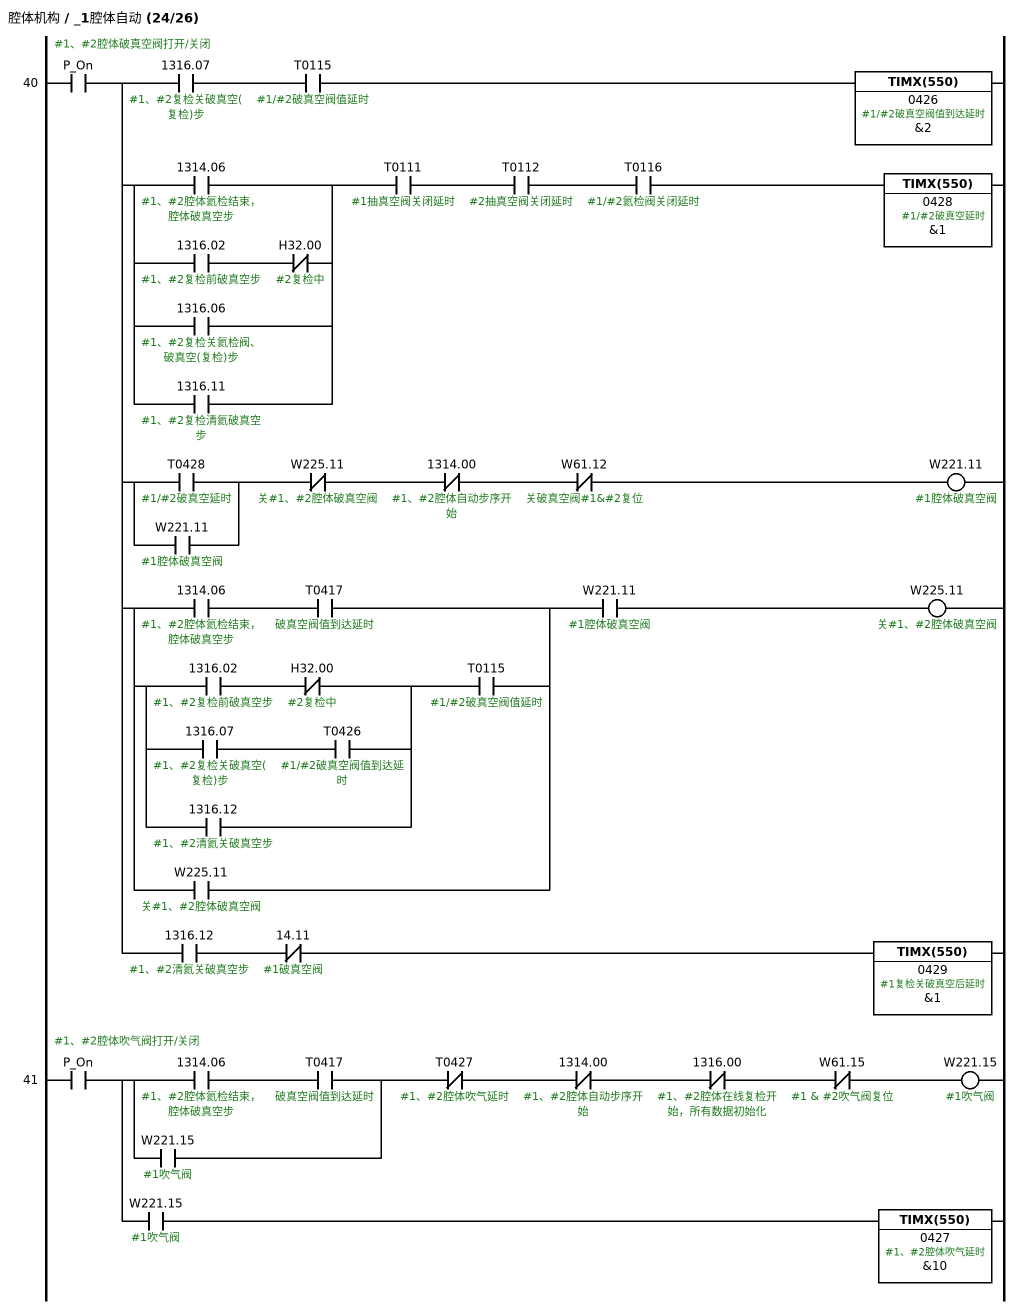
; [picture p264: 腔体机构 / _1腔体自动, rungs 40-41]
; rung 40: #1、#2腔体破真空阀打开/关闭
LD P_On
OUT TR0
AND 1316.07  ; #1、#2复检关破真空(复检)步
AND T0115  ; #1/#2破真空阀值延时
TIMX(550) 0426 &2  ; #1/#2破真空阀值到达延时
LD TR0
LD 1314.06  ; #1、#2腔体氦检结束，腔体破真空步
LD 1316.02  ; #1、#2复检前破真空步
ANDNOT H32.00  ; #2复检中
ORLD
OR 1316.06  ; #1、#2复检关氦检阀、破真空(复检)步
OR 1316.11  ; #1、#2复检清氦破真空步
ANDLD
AND T0111  ; #1抽真空阀关闭延时
AND T0112  ; #2抽真空阀关闭延时
AND T0116  ; #1/#2氦检阀关闭延时
TIMX(550) 0428 &1  ; #1/#2破真空延时
LD TR0
LD T0428  ; #1/#2破真空延时
OR W221.11  ; #1腔体破真空阀
ANDLD
ANDNOT W225.11  ; 关#1、#2腔体破真空阀
ANDNOT 1314.00  ; #1、#2腔体自动步序开始
ANDNOT W61.12  ; 关破真空阀#1&#2复位
OUT W221.11  ; #1腔体破真空阀
LD TR0
LD 1314.06  ; #1、#2腔体氦检结束，腔体破真空步
AND T0417  ; 破真空阀值到达延时
LD 1316.02  ; #1、#2复检前破真空步
ANDNOT H32.00  ; #2复检中
LD 1316.07  ; #1、#2复检关破真空(复检)步
AND T0426  ; #1/#2破真空阀值到达延时
ORLD
OR 1316.12  ; #1、#2清氦关破真空步
AND T0115  ; #1/#2破真空阀值延时
ORLD
OR W225.11  ; 关#1、#2腔体破真空阀
ANDLD
AND W221.11  ; #1腔体破真空阀
OUT W225.11  ; 关#1、#2腔体破真空阀
LD TR0
AND 1316.12  ; #1、#2清氦关破真空步
ANDNOT 14.11  ; #1破真空阀
TIMX(550) 0429 &1  ; #1复检关破真空后延时
; rung 41: #1、#2腔体吹气阀打开/关闭
LD P_On
OUT TR0
LD 1314.06  ; #1、#2腔体氦检结束，腔体破真空步
AND T0417  ; 破真空阀值到达延时
OR W221.15  ; #1吹气阀
ANDLD
ANDNOT T0427  ; #1、#2腔体吹气延时
ANDNOT 1314.00  ; #1、#2腔体自动步序开始
ANDNOT 1316.00  ; #1、#2腔体在线复检开始，所有数据初始化
ANDNOT W61.15  ; #1 & #2吹气阀复位
OUT W221.15  ; #1吹气阀
LD TR0
AND W221.15  ; #1吹气阀
TIMX(550) 0427 &10  ; #1、#2腔体吹气延时

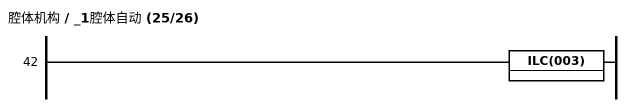
; rung 42
ILC(003)

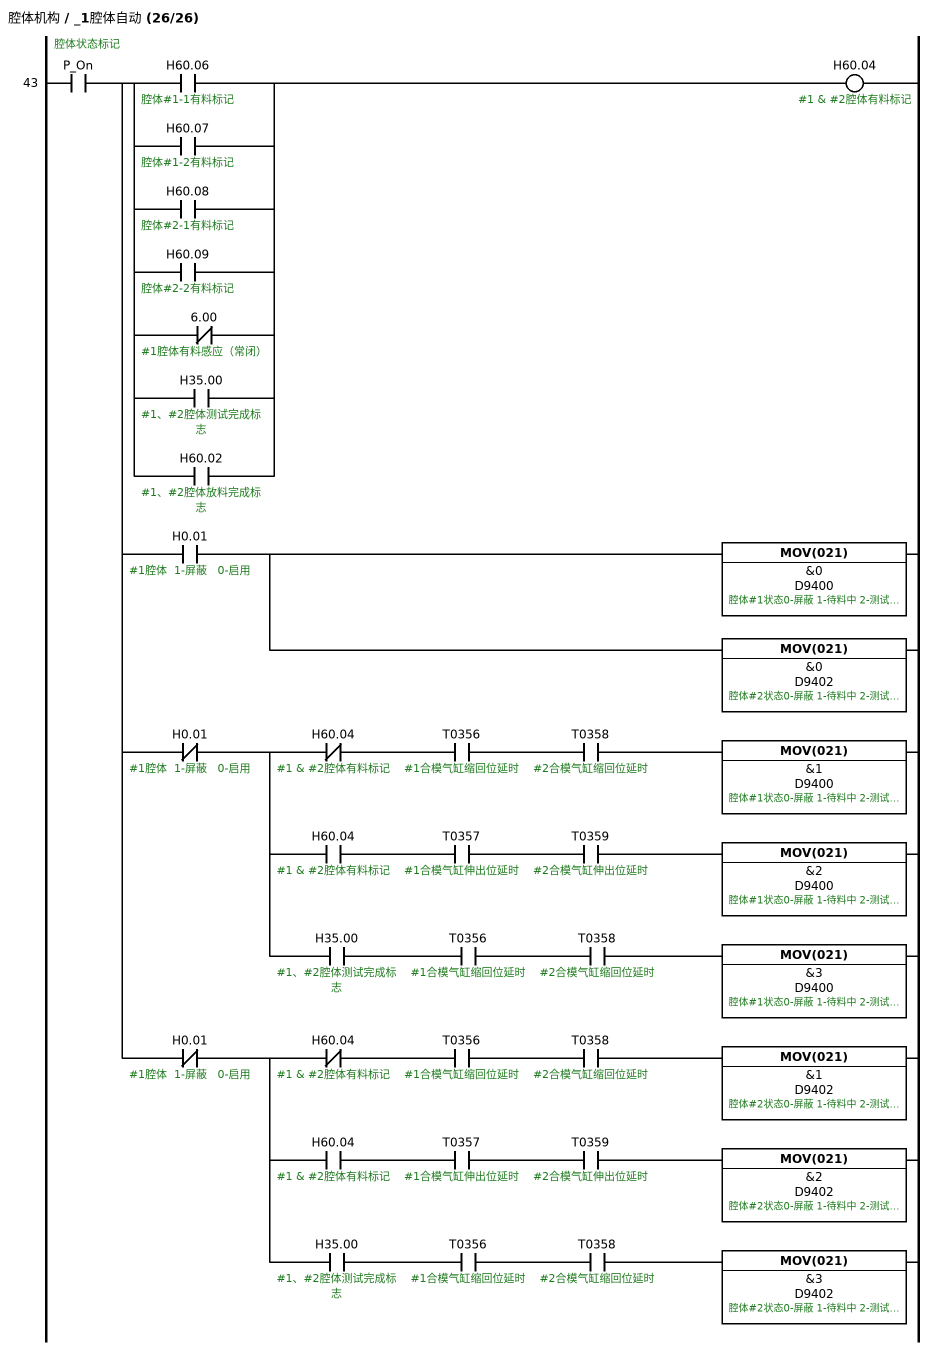
; rung 43: 腔体状态标记
LD P_On
OUT TR0
LD H60.06  ; 腔体#1-1有料标记
OR H60.07  ; 腔体#1-2有料标记
OR H60.08  ; 腔体#2-1有料标记
OR H60.09  ; 腔体#2-2有料标记
ORNOT 6.00  ; #1腔体有料感应（常闭）
OR H35.00  ; #1、#2腔体测试完成标志
OR H60.02  ; #1、#2腔体放料完成标志
ANDLD
OUT H60.04  ; #1 & #2腔体有料标记
LD TR0
AND H0.01  ; #1腔体  1-屏蔽   0-启用
MOV(021) &0 D9400  ; 腔体#1状态0-屏蔽 1-待料中 2-测试中 3-测试完成 4-在线复检
MOV(021) &0 D9402  ; 腔体#2状态0-屏蔽 1-待料中 2-测试中 3-测试完成 4-在线复检
LD TR0
ANDNOT H0.01  ; #1腔体  1-屏蔽   0-启用
OUT TR1
ANDNOT H60.04  ; #1 & #2腔体有料标记
AND T0356  ; #1合模气缸缩回位延时
AND T0358  ; #2合模气缸缩回位延时
MOV(021) &1 D9400  ; 腔体#1状态0-屏蔽 1-待料中 2-测试中 3-测试完成 4-在线复检
LD TR1
AND H60.04  ; #1 & #2腔体有料标记
AND T0357  ; #1合模气缸伸出位延时
AND T0359  ; #2合模气缸伸出位延时
MOV(021) &2 D9400  ; 腔体#1状态0-屏蔽 1-待料中 2-测试中 3-测试完成 4-在线复检
LD TR1
AND H35.00  ; #1、#2腔体测试完成标志
AND T0356  ; #1合模气缸缩回位延时
AND T0358  ; #2合模气缸缩回位延时
MOV(021) &3 D9400  ; 腔体#1状态0-屏蔽 1-待料中 2-测试中 3-测试完成 4-在线复检
LD TR0
ANDNOT H0.01  ; #1腔体  1-屏蔽   0-启用
OUT TR0
ANDNOT H60.04  ; #1 & #2腔体有料标记
AND T0356  ; #1合模气缸缩回位延时
AND T0358  ; #2合模气缸缩回位延时
MOV(021) &1 D9402  ; 腔体#2状态0-屏蔽 1-待料中 2-测试中 3-测试完成 4-在线复检
LD TR0
AND H60.04  ; #1 & #2腔体有料标记
AND T0357  ; #1合模气缸伸出位延时
AND T0359  ; #2合模气缸伸出位延时
MOV(021) &2 D9402  ; 腔体#2状态0-屏蔽 1-待料中 2-测试中 3-测试完成 4-在线复检
LD TR0
AND H35.00  ; #1、#2腔体测试完成标志
AND T0356  ; #1合模气缸缩回位延时
AND T0358  ; #2合模气缸缩回位延时
MOV(021) &3 D9402  ; 腔体#2状态0-屏蔽 1-待料中 2-测试中 3-测试完成 4-在线复检

### Section _2腔体自动

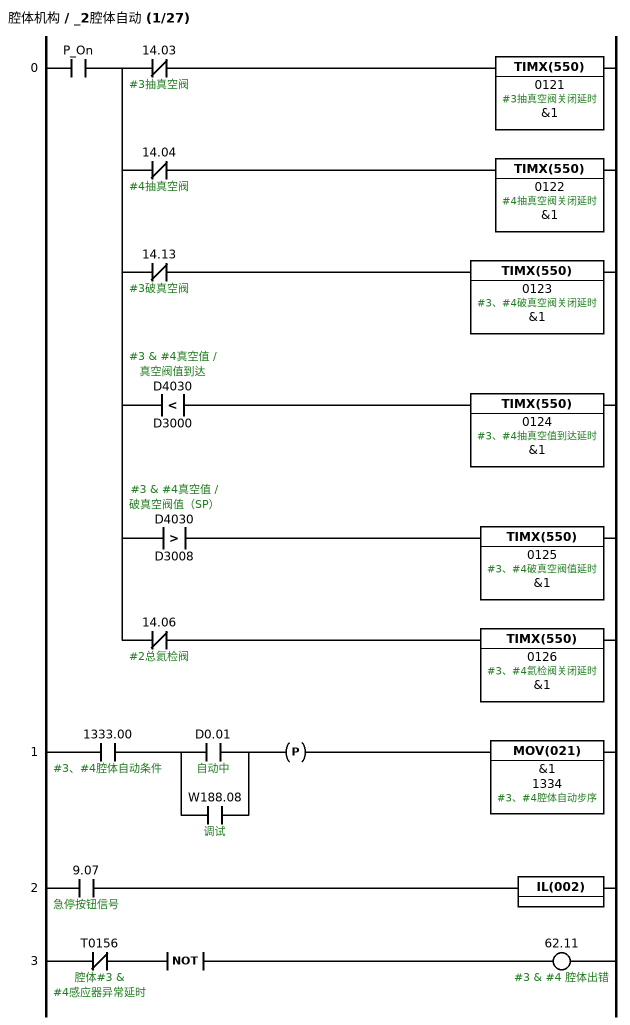
; rung 0
LD P_On
OUT TR0
ANDNOT 14.03  ; #3抽真空阀
TIMX(550) 0121 &1  ; #3抽真空阀关闭延时
LD TR0
ANDNOT 14.04  ; #4抽真空阀
TIMX(550) 0122 &1  ; #4抽真空阀关闭延时
LD TR0
ANDNOT 14.13  ; #3破真空阀
TIMX(550) 0123 &1  ; #3、#4破真空阀关闭延时
LD TR0
AND<F(331) D4030 D3000  ; #3 & #4真空值, 真空阀值到达
TIMX(550) 0124 &1  ; #3、#4抽真空值到达延时
LD TR0
AND>F(333) D4030 D3008  ; #3 & #4真空值, 破真空阀值（SP）
TIMX(550) 0125 &1  ; #3、#4破真空阀值延时
LD TR0
ANDNOT 14.06  ; #2总氦检阀
TIMX(550) 0126 &1  ; #3、#4氦检阀关闭延时
; rung 1
LD 1333.00  ; #3、#4腔体自动条件
LD D0.01  ; 自动中
OR W188.08  ; 调试
ANDLD
UP(521)
MOV(021) &1 1334  ; #3、#4腔体自动步序
; rung 2
LD 9.07  ; 急停按钮信号
IL(002)
; rung 3
LDNOT T0156  ; 腔体#3 & #4感应器异常延时
NOT(520)
OUT 62.11  ; #3 & #4 腔体出错

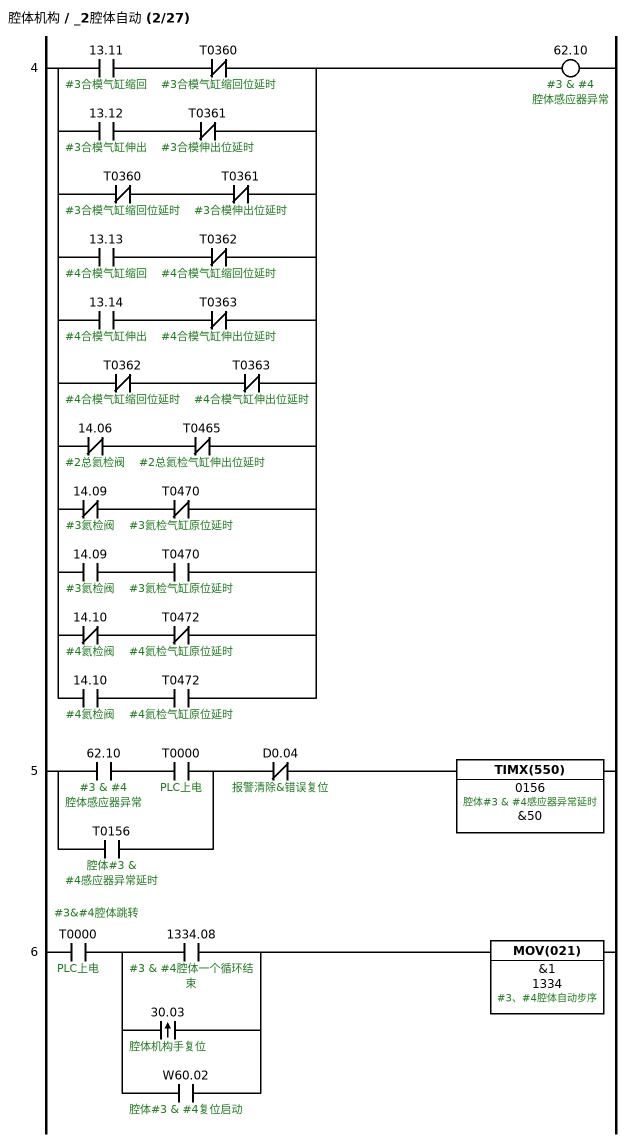
; rung 4
LD 13.11  ; #3合模气缸缩回
ANDNOT T0360  ; #3合模气缸缩回位延时
LD 13.12  ; #3合模气缸伸出
ANDNOT T0361  ; #3合模伸出位延时
ORLD
LDNOT T0360  ; #3合模气缸缩回位延时
ANDNOT T0361  ; #3合模伸出位延时
ORLD
LD 13.13  ; #4合模气缸缩回
ANDNOT T0362  ; #4合模气缸缩回位延时
ORLD
LD 13.14  ; #4合模气缸伸出
ANDNOT T0363  ; #4合模气缸伸出位延时
ORLD
LDNOT T0362  ; #4合模气缸缩回位延时
ANDNOT T0363  ; #4合模气缸伸出位延时
ORLD
LDNOT 14.06  ; #2总氦检阀
ANDNOT T0465  ; #2总氦检气缸伸出位延时
ORLD
LDNOT 14.09  ; #3氦检阀
ANDNOT T0470  ; #3氦检气缸原位延时
ORLD
LD 14.09  ; #3氦检阀
AND T0470  ; #3氦检气缸原位延时
ORLD
LDNOT 14.10  ; #4氦检阀
ANDNOT T0472  ; #4氦检气缸原位延时
ORLD
LD 14.10  ; #4氦检阀
AND T0472  ; #4氦检气缸原位延时
ORLD
OUT 62.10  ; #3 & #4 腔体感应器异常
; rung 5
LD 62.10  ; #3 & #4 腔体感应器异常
AND T0000  ; PLC上电
OR T0156  ; 腔体#3 & #4感应器异常延时
ANDNOT D0.04  ; 报警清除&错误复位
TIMX(550) 0156 &50  ; 腔体#3 & #4感应器异常延时
; rung 6: #3&#4腔体跳转
LD T0000  ; PLC上电
LD 1334.08  ; #3 & #4腔体一个循环结束
@OR 30.03  ; 腔体机构手复位
OR W60.02  ; 腔体#3 & #4复位启动
ANDLD
MOV(021) &1 1334  ; #3、#4腔体自动步序

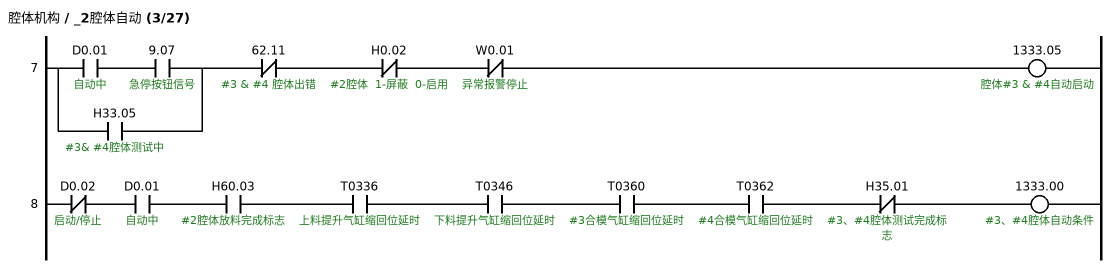
; rung 7
LD D0.01  ; 自动中
AND 9.07  ; 急停按钮信号
OR H33.05  ; #3& #4腔体测试中
ANDNOT 62.11  ; #3 & #4 腔体出错
ANDNOT H0.02  ; #2腔体  1-屏蔽  0-启用
ANDNOT W0.01  ; 异常报警停止
OUT 1333.05  ; 腔体#3 & #4自动启动
; rung 8
LDNOT D0.02  ; 启动/停止
AND D0.01  ; 自动中
AND H60.03  ; #2腔体放料完成标志
AND T0336  ; 上料提升气缸缩回位延时
AND T0346  ; 下料提升气缸缩回位延时
AND T0360  ; #3合模气缸缩回位延时
AND T0362  ; #4合模气缸缩回位延时
ANDNOT H35.01  ; #3、#4腔体测试完成标志
OUT 1333.00  ; #3、#4腔体自动条件

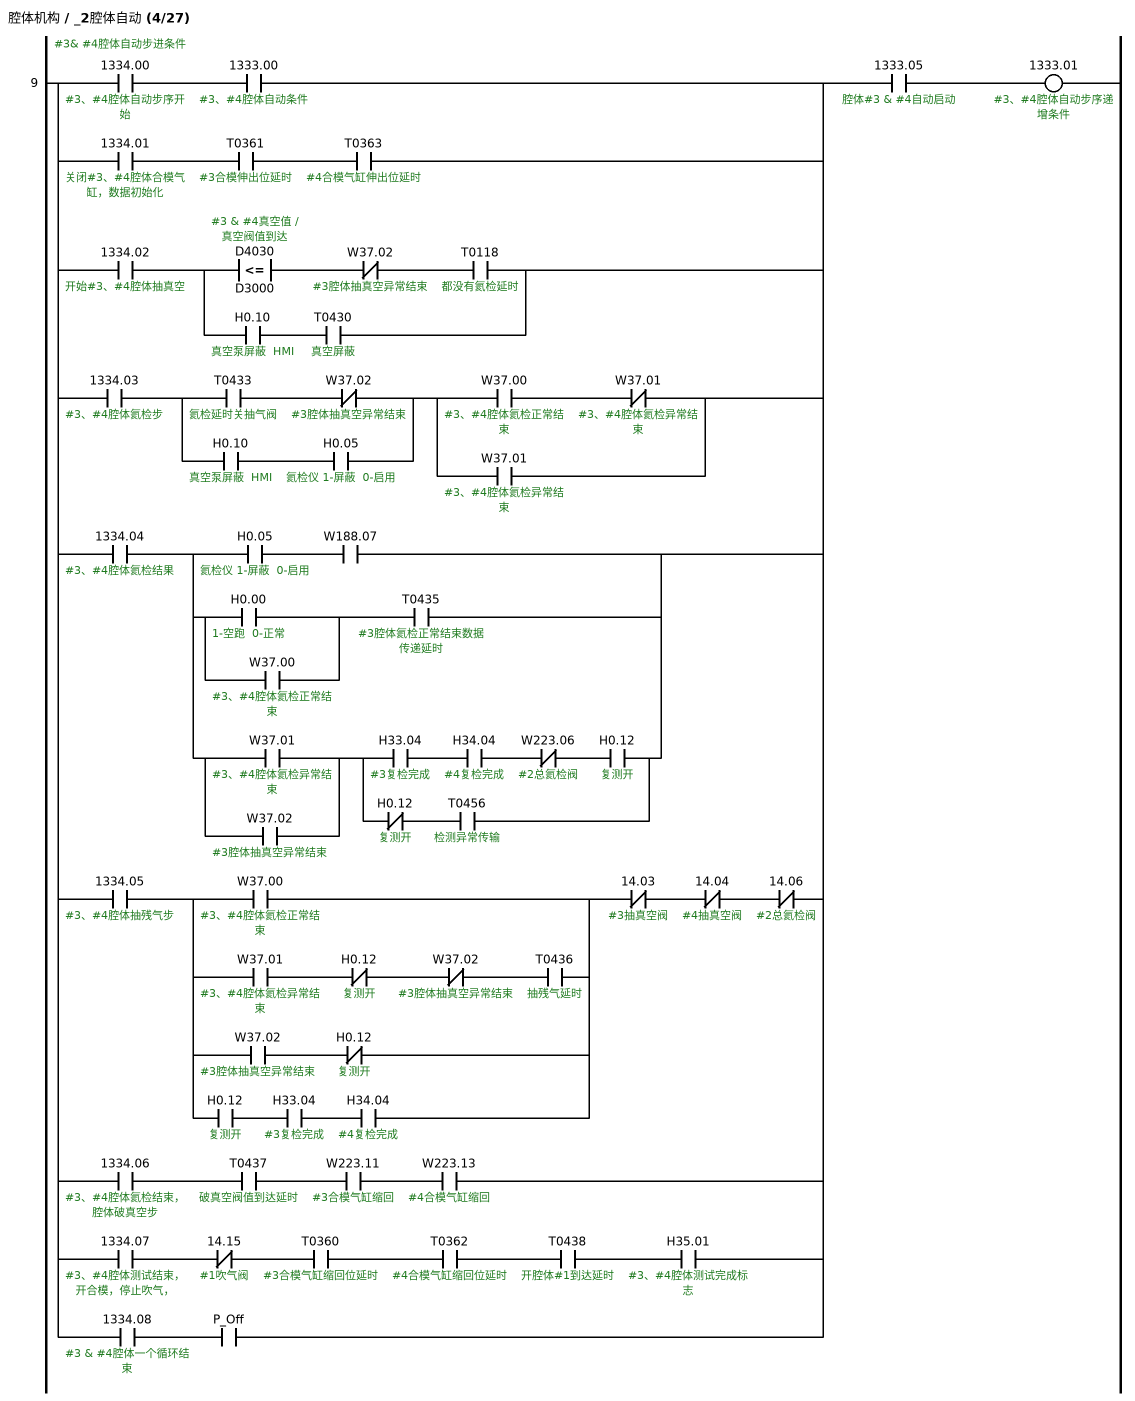
; rung 9: #3& #4腔体自动步进条件
LD 1334.00  ; #3、#4腔体自动步序开始
AND 1333.00  ; #3、#4腔体自动条件
LD 1334.01  ; 关闭#3、#4腔体合模气缸，数据初始化
AND T0361  ; #3合模伸出位延时
AND T0363  ; #4合模气缸伸出位延时
ORLD
LD 1334.02  ; 开始#3、#4腔体抽真空
LD<=F(332) D4030 D3000  ; #3 & #4真空值, 真空阀值到达
ANDNOT W37.02  ; #3腔体抽真空异常结束
AND T0118  ; 都没有氦检延时
LD H0.10  ; 真空泵屏蔽  HMI
AND T0430  ; 真空屏蔽
ORLD
ANDLD
ORLD
LD 1334.03  ; #3、#4腔体氦检步
LD T0433  ; 氦检延时关抽气阀
ANDNOT W37.02  ; #3腔体抽真空异常结束
LD H0.10  ; 真空泵屏蔽  HMI
AND H0.05  ; 氦检仪 1-屏蔽  0-启用
ORLD
ANDLD
LD W37.00  ; #3、#4腔体氦检正常结束
ANDNOT W37.01  ; #3、#4腔体氦检异常结束
OR W37.01  ; #3、#4腔体氦检异常结束
ANDLD
ORLD
LD 1334.04  ; #3、#4腔体氦检结果
LD H0.05  ; 氦检仪 1-屏蔽  0-启用
AND W188.07
LD H0.00  ; 1-空跑  0-正常
OR W37.00  ; #3、#4腔体氦检正常结束
AND T0435  ; #3腔体氦检正常结束数据传递延时
ORLD
LD W37.01  ; #3、#4腔体氦检异常结束
OR W37.02  ; #3腔体抽真空异常结束
LD H33.04  ; #3复检完成
AND H34.04  ; #4复检完成
ANDNOT W223.06  ; #2总氦检阀
AND H0.12  ; 复测开
LDNOT H0.12  ; 复测开
AND T0456  ; 检测异常传输
ORLD
ANDLD
ORLD
ANDLD
ORLD
LD 1334.05  ; #3、#4腔体抽残气步
LD W37.00  ; #3、#4腔体氦检正常结束
LD W37.01  ; #3、#4腔体氦检异常结束
ANDNOT H0.12  ; 复测开
ANDNOT W37.02  ; #3腔体抽真空异常结束
AND T0436  ; 抽残气延时
ORLD
LD W37.02  ; #3腔体抽真空异常结束
ANDNOT H0.12  ; 复测开
ORLD
LD H0.12  ; 复测开
AND H33.04  ; #3复检完成
AND H34.04  ; #4复检完成
ORLD
ANDLD
ANDNOT 14.03  ; #3抽真空阀
ANDNOT 14.04  ; #4抽真空阀
ANDNOT 14.06  ; #2总氦检阀
ORLD
LD 1334.06  ; #3、#4腔体氦检结束，腔体破真空步
AND T0437  ; 破真空阀值到达延时
AND W223.11  ; #3合模气缸缩回
AND W223.13  ; #4合模气缸缩回
ORLD
LD 1334.07  ; #3、#4腔体测试结束，开合模，停止吹气，
ANDNOT 14.15  ; #1吹气阀
AND T0360  ; #3合模气缸缩回位延时
AND T0362  ; #4合模气缸缩回位延时
AND T0438  ; 开腔体#1到达延时
AND H35.01  ; #3、#4腔体测试完成标志
ORLD
LD 1334.08  ; #3 & #4腔体一个循环结束
AND P_Off
ORLD
AND 1333.05  ; 腔体#3 & #4自动启动
OUT 1333.01  ; #3、#4腔体自动步序递增条件

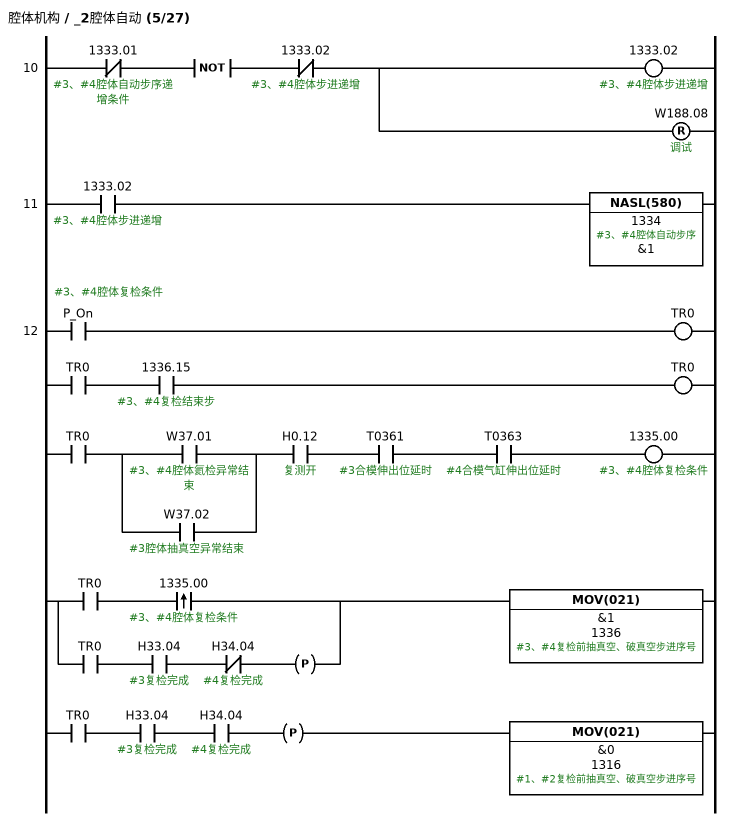
; rung 10
LDNOT 1333.01  ; #3、#4腔体自动步序递增条件
NOT(520)
ANDNOT 1333.02  ; #3、#4腔体步进递增
OUT 1333.02  ; #3、#4腔体步进递增
RSET W188.08  ; 调试
; rung 11
LD 1333.02  ; #3、#4腔体步进递增
NASL(580) 1334 &1  ; #3、#4腔体自动步序
; rung 12: #3、#4腔体复检条件
LD P_On
OUT TR0
LD W37.01  ; #3、#4腔体氦检异常结束
OR W37.02  ; #3腔体抽真空异常结束
ANDLD
AND H0.12  ; 复测开
AND T0361  ; #3合模伸出位延时
AND T0363  ; #4合模气缸伸出位延时
OUT 1335.00  ; #3、#4腔体复检条件
LD TR0
@AND 1335.00  ; #3、#4腔体复检条件
LD TR0
AND 1336.15  ; #3、#4复检结束步
OUT TR0
AND H33.04  ; #3复检完成
ANDNOT H34.04  ; #4复检完成
UP(521)
ORLD
MOV(021) &1 1336  ; #3、#4复检前抽真空、破真空步进序号
LD TR0
AND H33.04  ; #3复检完成
AND H34.04  ; #4复检完成
UP(521)
MOV(021) &0 1316  ; #1、#2复检前抽真空、破真空步进序号

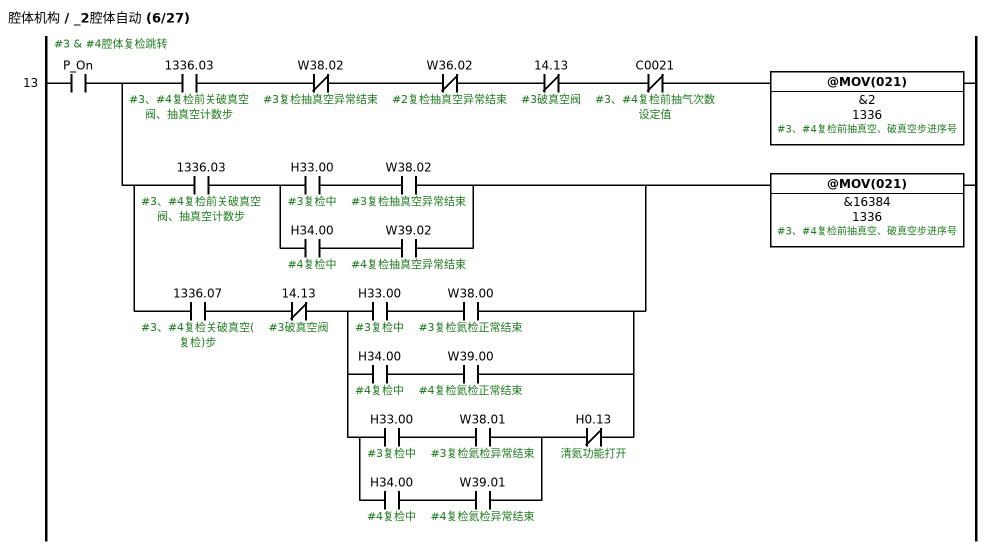
; rung 13: #3 & #4腔体复检跳转
LD P_On
OUT TR0
AND 1336.03  ; #3、#4复检前关破真空阀、抽真空计数步
ANDNOT W38.02  ; #3复检抽真空异常结束
ANDNOT W36.02  ; #2复检抽真空异常结束
ANDNOT 14.13  ; #3破真空阀
ANDNOT C0021  ; #3、#4复检前抽气次数设定值
@MOV(021) &2 1336  ; #3、#4复检前抽真空、破真空步进序号
LD TR0
LD 1336.03  ; #3、#4复检前关破真空阀、抽真空计数步
LD H33.00  ; #3复检中
AND W38.02  ; #3复检抽真空异常结束
LD H34.00  ; #4复检中
AND W39.02  ; #4复检抽真空异常结束
ORLD
ANDLD
LD 1336.07  ; #3、#4复检关破真空(复检)步
ANDNOT 14.13  ; #3破真空阀
LD H33.00  ; #3复检中
AND W38.00  ; #3复检氦检正常结束
LD H34.00  ; #4复检中
AND W39.00  ; #4复检氦检正常结束
ORLD
LD H33.00  ; #3复检中
AND W38.01  ; #3复检氦检异常结束
LD H34.00  ; #4复检中
AND W39.01  ; #4复检氦检异常结束
ORLD
ANDNOT H0.13  ; 清氦功能打开
ORLD
ANDLD
ORLD
ANDLD
@MOV(021) &16384 1336  ; #3、#4复检前抽真空、破真空步进序号

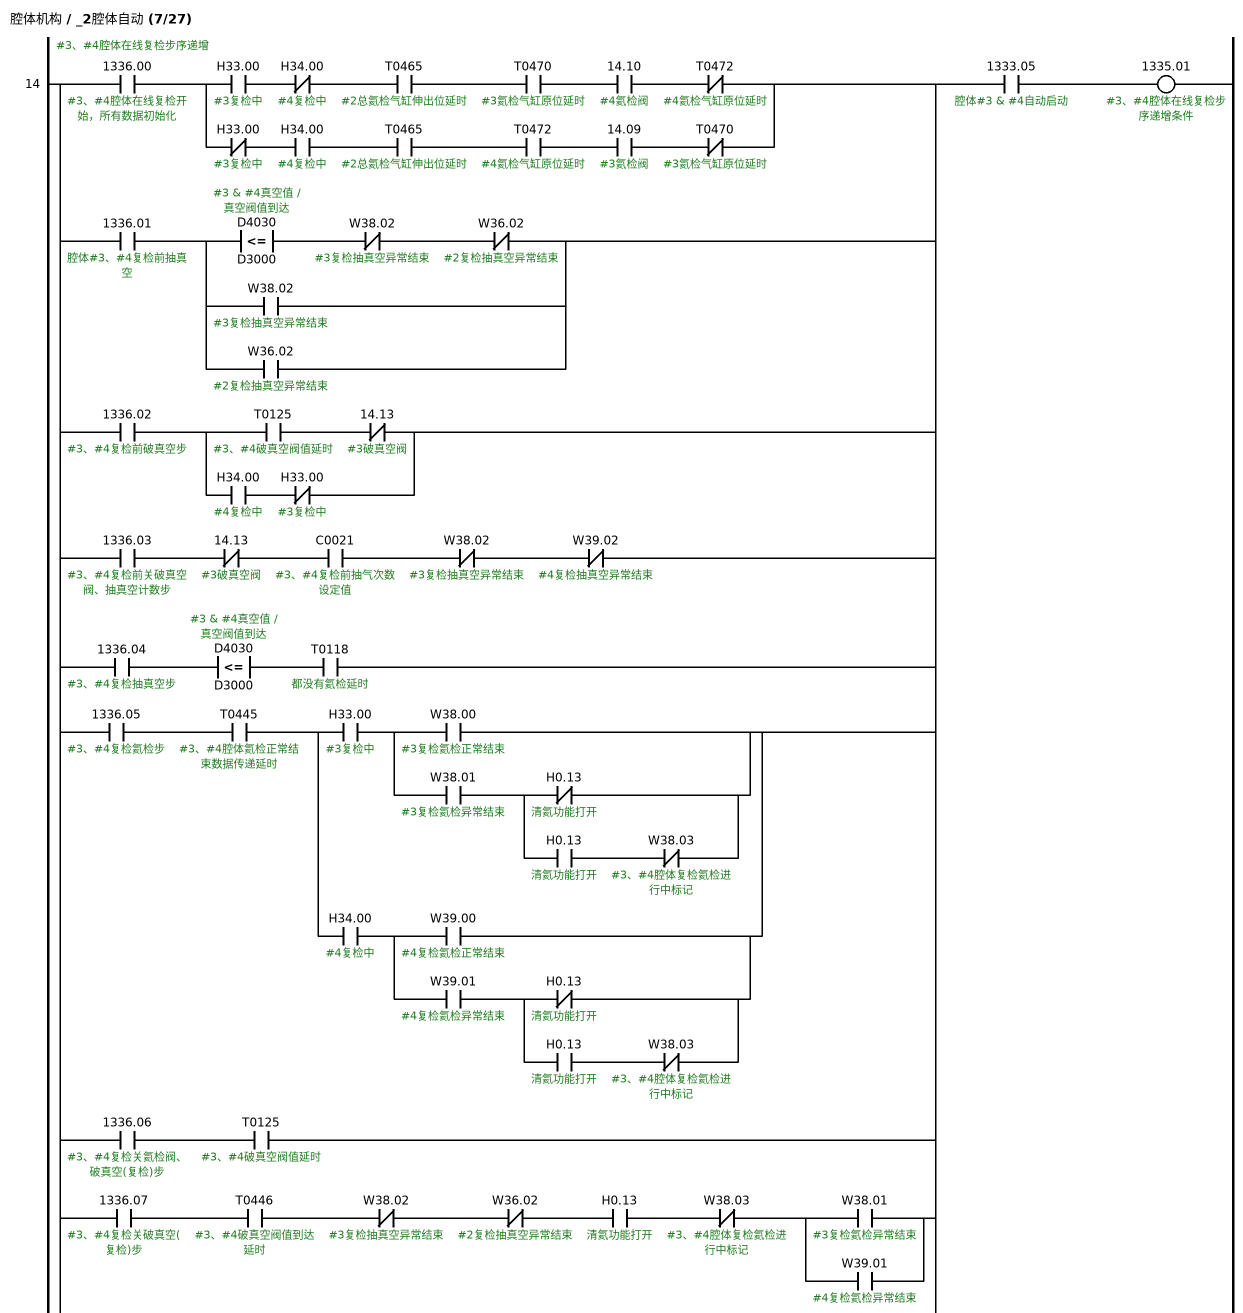

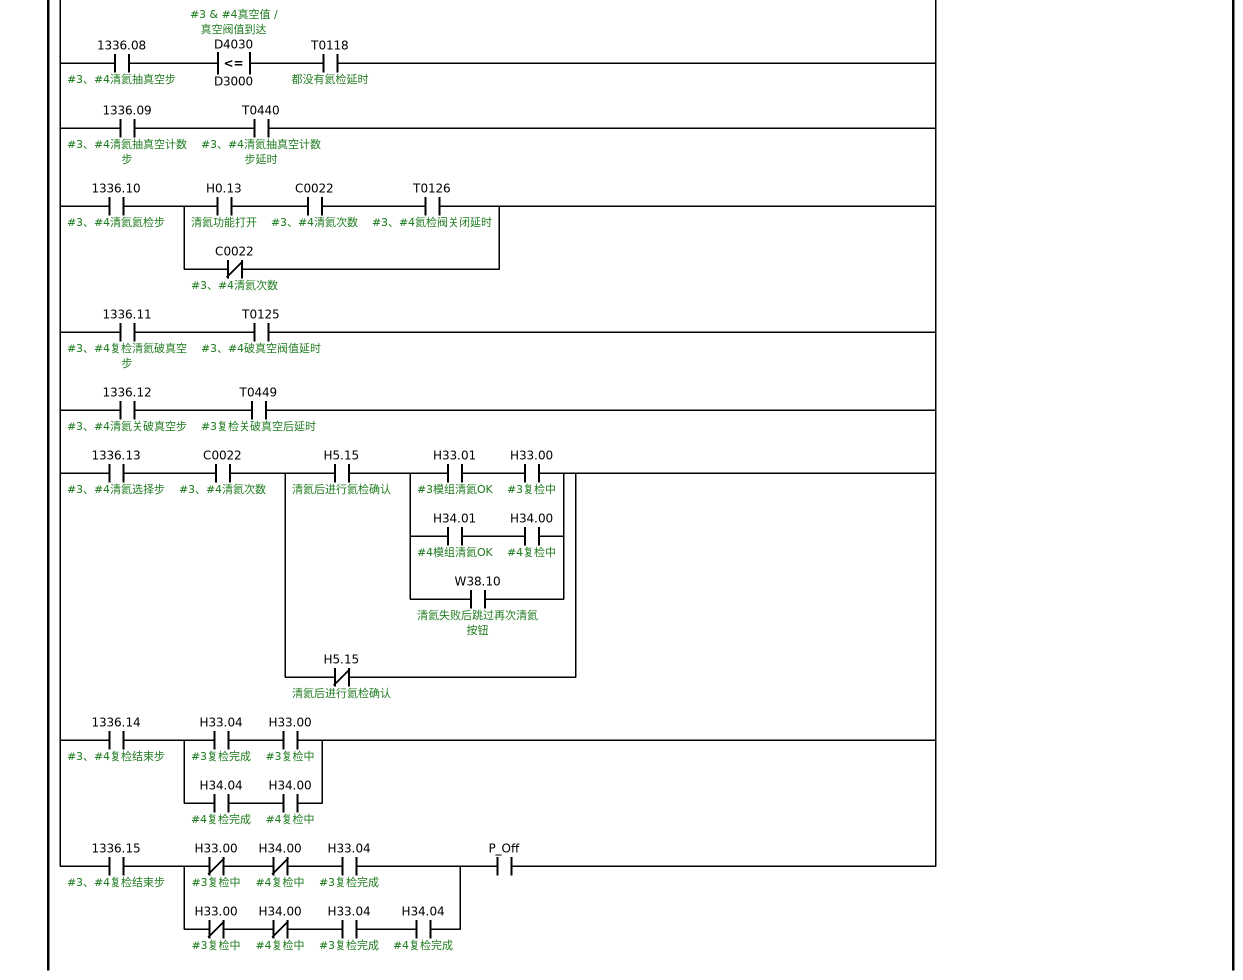
; rung 14: #3、#4腔体在线复检步序递增
LD 1336.00  ; #3、#4腔体在线复检开始，所有数据初始化
LD H33.00  ; #3复检中
ANDNOT H34.00  ; #4复检中
AND T0465  ; #2总氦检气缸伸出位延时
AND T0470  ; #3氦检气缸原位延时
AND 14.10  ; #4氦检阀
ANDNOT T0472  ; #4氦检气缸原位延时
LDNOT H33.00  ; #3复检中
AND H34.00  ; #4复检中
AND T0465  ; #2总氦检气缸伸出位延时
AND T0472  ; #4氦检气缸原位延时
AND 14.09  ; #3氦检阀
ANDNOT T0470  ; #3氦检气缸原位延时
ORLD
ANDLD
LD 1336.01  ; 腔体#3、#4复检前抽真空
LD<=F(332) D4030 D3000  ; #3 & #4真空值, 真空阀值到达
ANDNOT W38.02  ; #3复检抽真空异常结束
ANDNOT W36.02  ; #2复检抽真空异常结束
OR W38.02  ; #3复检抽真空异常结束
OR W36.02  ; #2复检抽真空异常结束
ANDLD
ORLD
LD 1336.02  ; #3、#4复检前破真空步
LD T0125  ; #3、#4破真空阀值延时
ANDNOT 14.13  ; #3破真空阀
LD H34.00  ; #4复检中
ANDNOT H33.00  ; #3复检中
ORLD
ANDLD
ORLD
LD 1336.03  ; #3、#4复检前关破真空阀、抽真空计数步
ANDNOT 14.13  ; #3破真空阀
AND C0021  ; #3、#4复检前抽气次数设定值
ANDNOT W38.02  ; #3复检抽真空异常结束
ANDNOT W39.02  ; #4复检抽真空异常结束
ORLD
LD 1336.04  ; #3、#4复检抽真空步
AND<=F(332) D4030 D3000  ; #3 & #4真空值, 真空阀值到达
AND T0118  ; 都没有氦检延时
ORLD
LD 1336.05  ; #3、#4复检氦检步
AND T0445  ; #3、#4腔体氦检正常结束数据传递延时
LD H33.00  ; #3复检中
LD W38.00  ; #3复检氦检正常结束
LD W38.01  ; #3复检氦检异常结束
LDNOT H0.13  ; 清氦功能打开
LD H0.13  ; 清氦功能打开
ANDNOT W38.03  ; #3、#4腔体复检氦检进行中标记
ORLD
ANDLD
ORLD
ANDLD
LD H34.00  ; #4复检中
LD W39.00  ; #4复检氦检正常结束
LD W39.01  ; #4复检氦检异常结束
LDNOT H0.13  ; 清氦功能打开
LD H0.13  ; 清氦功能打开
ANDNOT W38.03  ; #3、#4腔体复检氦检进行中标记
ORLD
ANDLD
ORLD
ANDLD
ORLD
ANDLD
ORLD
LD 1336.06  ; #3、#4复检关氦检阀、破真空(复检)步
AND T0125  ; #3、#4破真空阀值延时
ORLD
LD 1336.07  ; #3、#4复检关破真空(复检)步
AND T0446  ; #3、#4破真空阀值到达延时
ANDNOT W38.02  ; #3复检抽真空异常结束
ANDNOT W36.02  ; #2复检抽真空异常结束
AND H0.13  ; 清氦功能打开
ANDNOT W38.03  ; #3、#4腔体复检氦检进行中标记
LD W38.01  ; #3复检氦检异常结束
OR W39.01  ; #4复检氦检异常结束
ANDLD
ORLD
LD 1336.08  ; #3、#4清氦抽真空步
AND<=F(332) D4030 D3000  ; #3 & #4真空值, 真空阀值到达
AND T0118  ; 都没有氦检延时
ORLD
LD 1336.09  ; #3、#4清氦抽真空计数步
AND T0440  ; #3、#4清氦抽真空计数步延时
ORLD
LD 1336.10  ; #3、#4清氦氦检步
LD H0.13  ; 清氦功能打开
AND C0022  ; #3、#4清氦次数
AND T0126  ; #3、#4氦检阀关闭延时
ORNOT C0022  ; #3、#4清氦次数
ANDLD
ORLD
LD 1336.11  ; #3、#4复检清氦破真空步
AND T0125  ; #3、#4破真空阀值延时
ORLD
LD 1336.12  ; #3、#4清氦关破真空步
AND T0449  ; #3复检关破真空后延时
ORLD
LD 1336.13  ; #3、#4清氦选择步
AND C0022  ; #3、#4清氦次数
LD H5.15  ; 清氦后进行氦检确认
LD H33.01  ; #3模组清氦OK
AND H33.00  ; #3复检中
LD H34.01  ; #4模组清氦OK
AND H34.00  ; #4复检中
ORLD
OR W38.10  ; 清氦失败后跳过再次清氦按钮
ANDLD
ORNOT H5.15  ; 清氦后进行氦检确认
ANDLD
ORLD
LD 1336.14  ; #3、#4复检结束步
LD H33.04  ; #3复检完成
AND H33.00  ; #3复检中
LD H34.04  ; #4复检完成
AND H34.00  ; #4复检中
ORLD
ANDLD
ORLD
LD 1336.15  ; #3、#4复检结束步
LDNOT H33.00  ; #3复检中
ANDNOT H34.00  ; #4复检中
AND H33.04  ; #3复检完成
LDNOT H33.00  ; #3复检中
ANDNOT H34.00  ; #4复检中
AND H33.04  ; #3复检完成
AND H34.04  ; #4复检完成
ORLD
ANDLD
AND P_Off
ORLD
AND 1333.05  ; 腔体#3 & #4自动启动
OUT 1335.01  ; #3、#4腔体在线复检步序递增条件

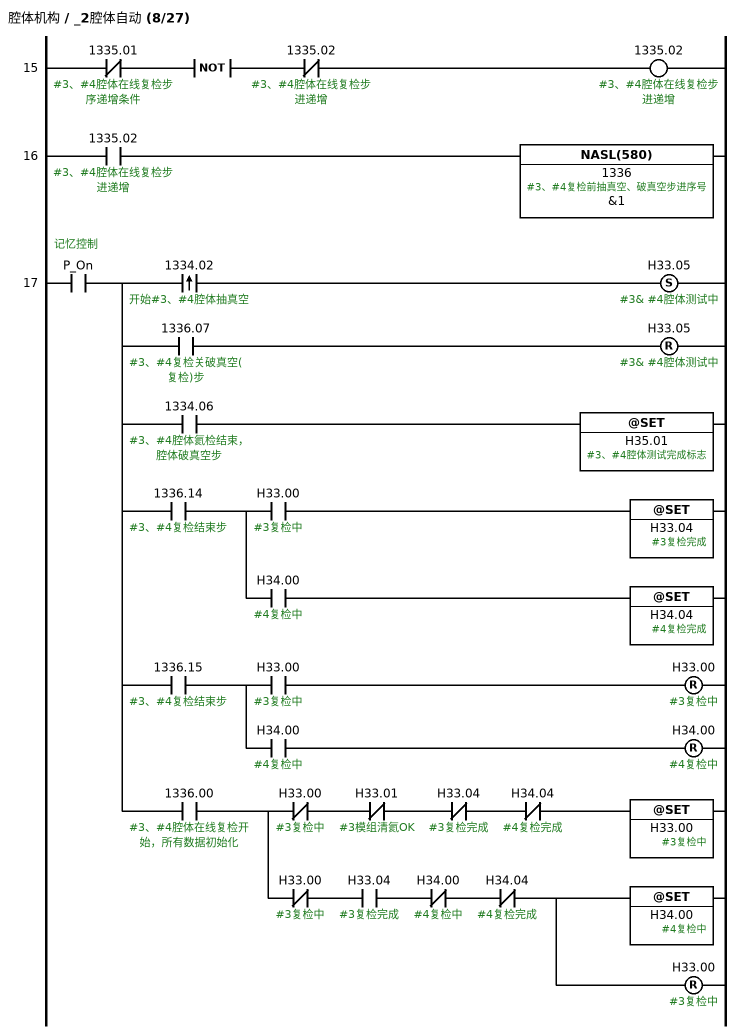
; rung 15
LDNOT 1335.01  ; #3、#4腔体在线复检步序递增条件
NOT(520)
ANDNOT 1335.02  ; #3、#4腔体在线复检步进递增
OUT 1335.02  ; #3、#4腔体在线复检步进递增
; rung 16
LD 1335.02  ; #3、#4腔体在线复检步进递增
NASL(580) 1336 &1  ; #3、#4复检前抽真空、破真空步进序号
; rung 17: 记忆控制
LD P_On
OUT TR0
@AND 1334.02  ; 开始#3、#4腔体抽真空
SET H33.05  ; #3& #4腔体测试中
LD TR0
AND 1336.07  ; #3、#4复检关破真空(复检)步
RSET H33.05  ; #3& #4腔体测试中
LD TR0
AND 1334.06  ; #3、#4腔体氦检结束，腔体破真空步
@SET H35.01  ; #3、#4腔体测试完成标志
LD TR0
AND 1336.14  ; #3、#4复检结束步
OUT TR1
AND H33.00  ; #3复检中
@SET H33.04  ; #3复检完成
LD TR1
AND H34.00  ; #4复检中
@SET H34.04  ; #4复检完成
LD TR0
AND 1336.15  ; #3、#4复检结束步
OUT TR1
AND H33.00  ; #3复检中
RSET H33.00  ; #3复检中
LD TR1
AND H34.00  ; #4复检中
RSET H34.00  ; #4复检中
LD TR0
AND 1336.00  ; #3、#4腔体在线复检开始，所有数据初始化
OUT TR0
ANDNOT H33.00  ; #3复检中
ANDNOT H33.01  ; #3模组清氦OK
ANDNOT H33.04  ; #3复检完成
ANDNOT H34.04  ; #4复检完成
@SET H33.00  ; #3复检中
LD TR0
ANDNOT H33.00  ; #3复检中
AND H33.04  ; #3复检完成
ANDNOT H34.00  ; #4复检中
ANDNOT H34.04  ; #4复检完成
@SET H34.00  ; #4复检中
RSET H33.00  ; #3复检中

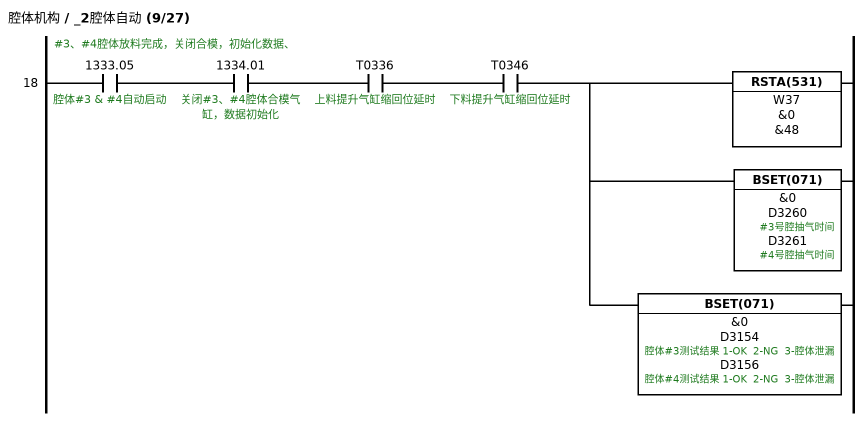
; rung 18: #3、#4腔体放料完成，关闭合模，初始化数据、
LD 1333.05  ; 腔体#3 & #4自动启动
AND 1334.01  ; 关闭#3、#4腔体合模气缸，数据初始化
AND T0336  ; 上料提升气缸缩回位延时
AND T0346  ; 下料提升气缸缩回位延时
RSTA(531) W37 &0 &48
BSET(071) &0 D3260 D3261  ; #3号腔抽气时间, #4号腔抽气时间
BSET(071) &0 D3154 D3156  ; 腔体#3测试结果 1-OK  2-NG  3-腔体泄漏, 腔体#4测试结果 1-OK  2-NG  3-腔体泄漏

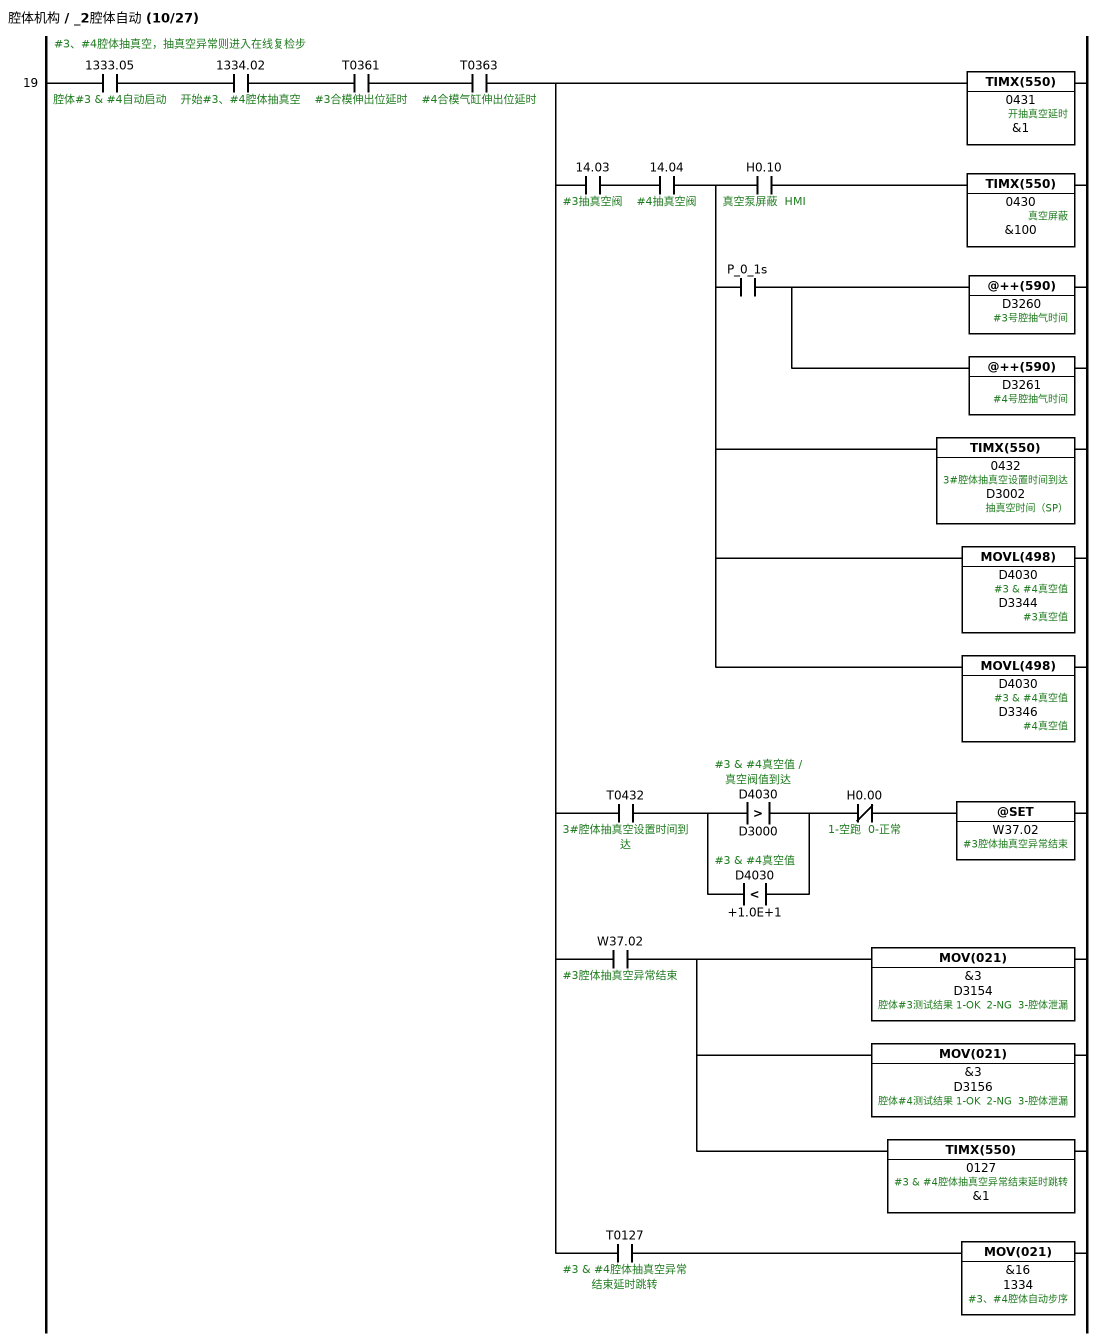
; rung 19: #3、#4腔体抽真空，抽真空异常则进入在线复检步
LD 1333.05  ; 腔体#3 & #4自动启动
AND 1334.02  ; 开始#3、#4腔体抽真空
AND T0361  ; #3合模伸出位延时
AND T0363  ; #4合模气缸伸出位延时
OUT TR0
TIMX(550) 0431 &1  ; 开抽真空延时
AND 14.03  ; #3抽真空阀
AND 14.04  ; #4抽真空阀
OUT TR1
AND H0.10  ; 真空泵屏蔽  HMI
TIMX(550) 0430 &100  ; 真空屏蔽
LD TR1
AND P_0_1s
@++(590) D3260  ; #3号腔抽气时间
@++(590) D3261  ; #4号腔抽气时间
LD TR1
TIMX(550) 0432 D3002  ; 抽真空时间（SP）, 3#腔体抽真空设置时间到达
MOVL(498) D4030 D3344  ; #3 & #4真空值, #3真空值
MOVL(498) D4030 D3346  ; #3 & #4真空值, #4真空值
LD TR0
AND T0432  ; 3#腔体抽真空设置时间到达
LD>F(333) D4030 D3000  ; #3 & #4真空值, 真空阀值到达
OR<F(331) D4030 +1.0E+1  ; #3 & #4真空值
ANDLD
ANDNOT H0.00  ; 1-空跑  0-正常
@SET W37.02  ; #3腔体抽真空异常结束
LD TR0
AND W37.02  ; #3腔体抽真空异常结束
MOV(021) &3 D3154  ; 腔体#3测试结果 1-OK  2-NG  3-腔体泄漏
MOV(021) &3 D3156  ; 腔体#4测试结果 1-OK  2-NG  3-腔体泄漏
TIMX(550) 0127 &1  ; #3 & #4腔体抽真空异常结束延时跳转
LD TR0
AND T0127  ; #3 & #4腔体抽真空异常结束延时跳转
MOV(021) &16 1334  ; #3、#4腔体自动步序

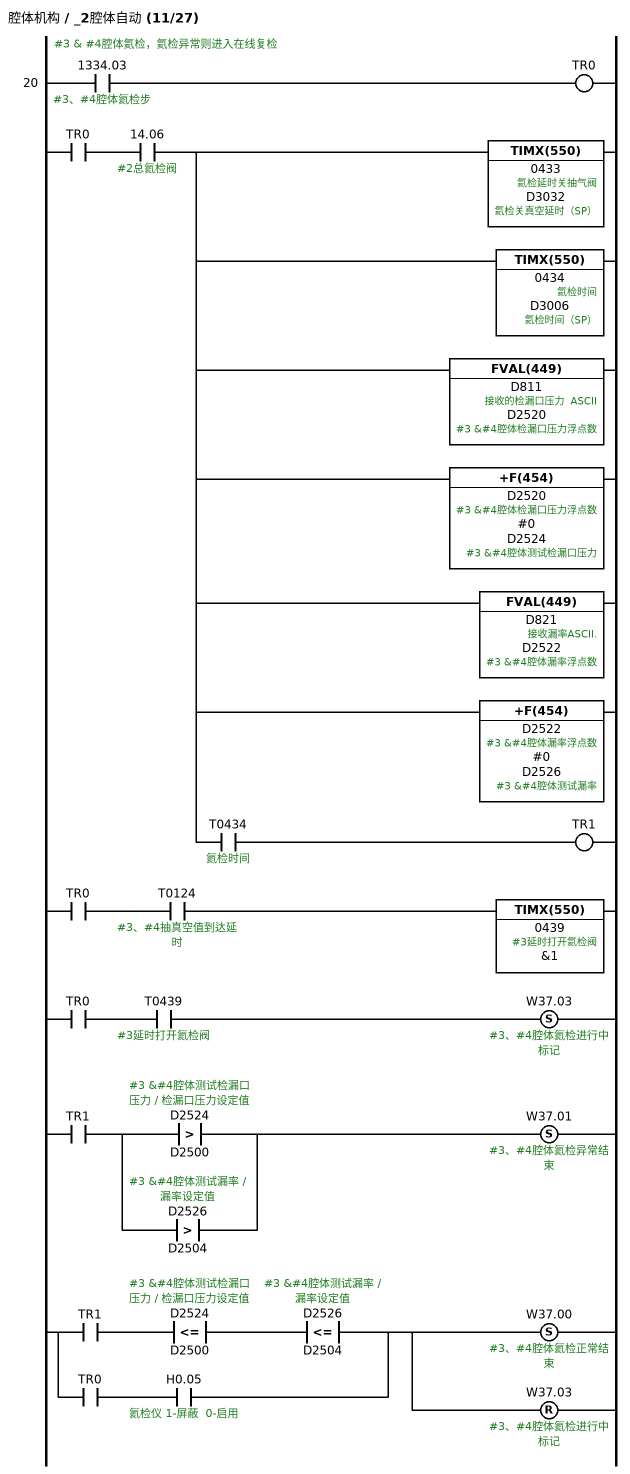
; rung 20: #3 & #4腔体氦检，氦检异常则进入在线复检
LD 1334.03  ; #3、#4腔体氦检步
OUT TR0
AND T0124  ; #3、#4抽真空值到达延时
TIMX(550) 0439 &1  ; #3延时打开氦检阀
LD TR0
AND T0439  ; #3延时打开氦检阀
SET W37.03  ; #3、#4腔体氦检进行中标记
LD TR0
AND 14.06  ; #2总氦检阀
TIMX(550) 0433 D3032  ; 氦检关真空延时（SP）, 氦检延时关抽气阀
TIMX(550) 0434 D3006  ; 氦检时间（SP）, 氦检时间
FVAL(449) D811 D2520  ; 接收的检漏口压力  ASCII, #3 &#4腔体检漏口压力浮点数
+F(454) D2520 #0 D2524  ; #3 &#4腔体检漏口压力浮点数, #3 &#4腔体测试检漏口压力
FVAL(449) D821 D2522  ; 接收漏率ASCII., #3 &#4腔体漏率浮点数
+F(454) D2522 #0 D2526  ; #3 &#4腔体漏率浮点数, #3 &#4腔体测试漏率
AND T0434  ; 氦检时间
OUT TR1
LD>F(333) D2524 D2500  ; #3 &#4腔体测试检漏口压力, 检漏口压力设定值
OR>F(333) D2526 D2504  ; #3 &#4腔体测试漏率, 漏率设定值
ANDLD
SET W37.01  ; #3、#4腔体氦检异常结束
LD TR1
AND<=F(332) D2524 D2500  ; #3 &#4腔体测试检漏口压力, 检漏口压力设定值
AND<=F(332) D2526 D2504  ; #3 &#4腔体测试漏率, 漏率设定值
LD TR0
AND H0.05  ; 氦检仪 1-屏蔽  0-启用
ORLD
SET W37.00  ; #3、#4腔体氦检正常结束
RSET W37.03  ; #3、#4腔体氦检进行中标记

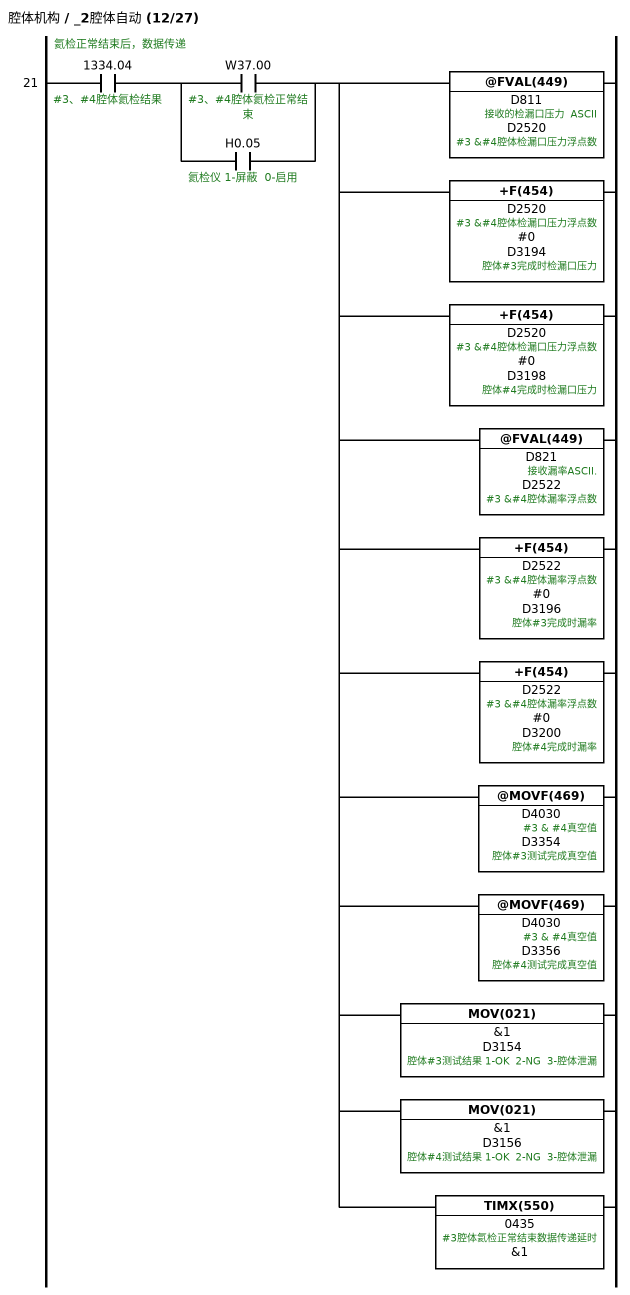
; rung 21: 氦检正常结束后，数据传递
LD 1334.04  ; #3、#4腔体氦检结果
LD W37.00  ; #3、#4腔体氦检正常结束
OR H0.05  ; 氦检仪 1-屏蔽  0-启用
ANDLD
@FVAL(449) D811 D2520  ; 接收的检漏口压力  ASCII, #3 &#4腔体检漏口压力浮点数
+F(454) D2520 #0 D3194  ; #3 &#4腔体检漏口压力浮点数, 腔体#3完成时检漏口压力
+F(454) D2520 #0 D3198  ; #3 &#4腔体检漏口压力浮点数, 腔体#4完成时检漏口压力
@FVAL(449) D821 D2522  ; 接收漏率ASCII., #3 &#4腔体漏率浮点数
+F(454) D2522 #0 D3196  ; #3 &#4腔体漏率浮点数, 腔体#3完成时漏率
+F(454) D2522 #0 D3200  ; #3 &#4腔体漏率浮点数, 腔体#4完成时漏率
@MOVF(469) D4030 D3354  ; #3 & #4真空值, 腔体#3测试完成真空值
@MOVF(469) D4030 D3356  ; #3 & #4真空值, 腔体#4测试完成真空值
MOV(021) &1 D3154  ; 腔体#3测试结果 1-OK  2-NG  3-腔体泄漏
MOV(021) &1 D3156  ; 腔体#4测试结果 1-OK  2-NG  3-腔体泄漏
TIMX(550) 0435 &1  ; #3腔体氦检正常结束数据传递延时

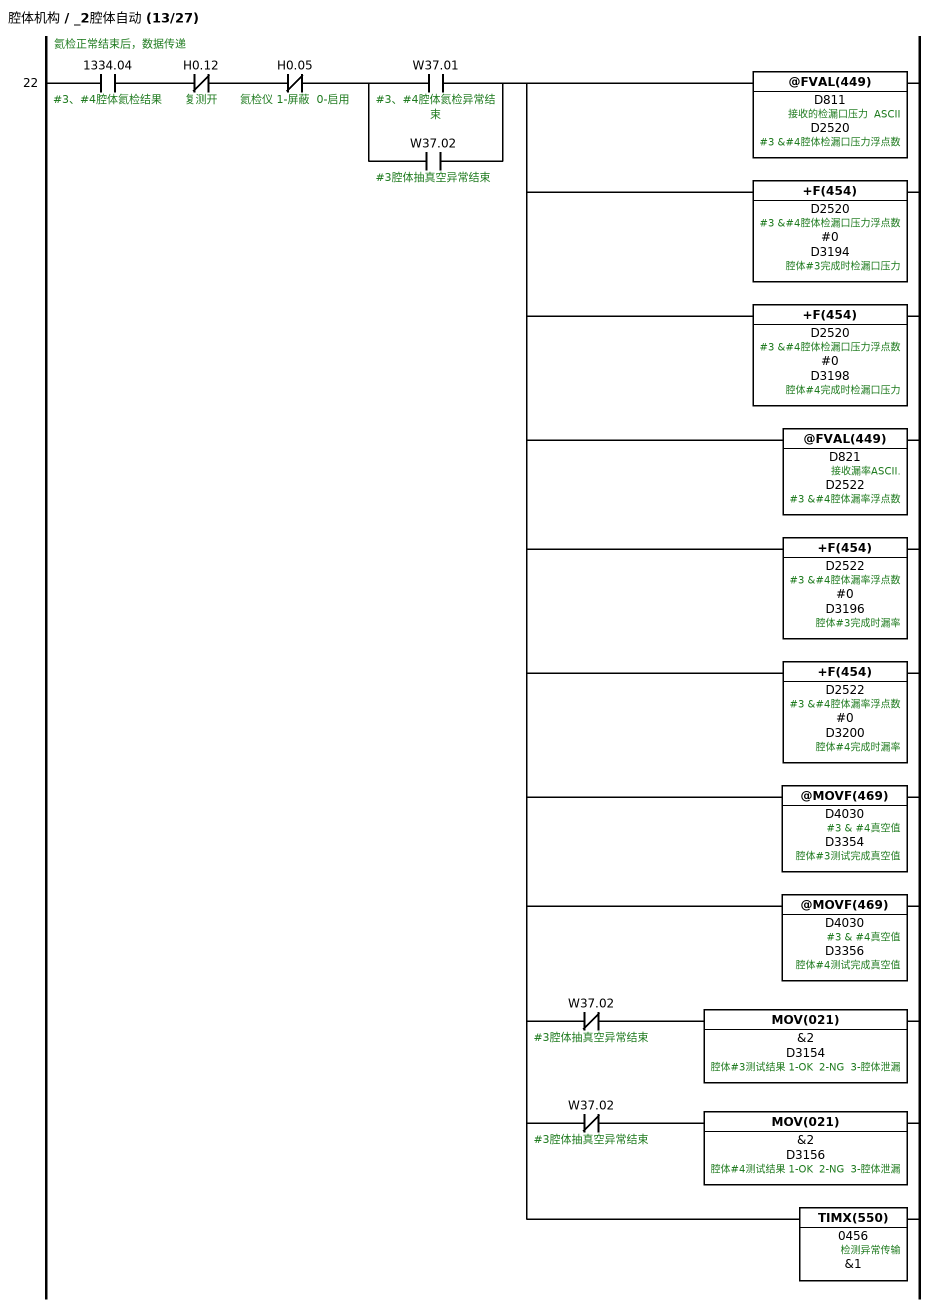
; rung 22: 氦检正常结束后，数据传递
LD 1334.04  ; #3、#4腔体氦检结果
ANDNOT H0.12  ; 复测开
ANDNOT H0.05  ; 氦检仪 1-屏蔽  0-启用
LD W37.01  ; #3、#4腔体氦检异常结束
OR W37.02  ; #3腔体抽真空异常结束
ANDLD
OUT TR0
@FVAL(449) D811 D2520  ; 接收的检漏口压力  ASCII, #3 &#4腔体检漏口压力浮点数
+F(454) D2520 #0 D3194  ; #3 &#4腔体检漏口压力浮点数, 腔体#3完成时检漏口压力
+F(454) D2520 #0 D3198  ; #3 &#4腔体检漏口压力浮点数, 腔体#4完成时检漏口压力
@FVAL(449) D821 D2522  ; 接收漏率ASCII., #3 &#4腔体漏率浮点数
+F(454) D2522 #0 D3196  ; #3 &#4腔体漏率浮点数, 腔体#3完成时漏率
+F(454) D2522 #0 D3200  ; #3 &#4腔体漏率浮点数, 腔体#4完成时漏率
@MOVF(469) D4030 D3354  ; #3 & #4真空值, 腔体#3测试完成真空值
@MOVF(469) D4030 D3356  ; #3 & #4真空值, 腔体#4测试完成真空值
ANDNOT W37.02  ; #3腔体抽真空异常结束
MOV(021) &2 D3154  ; 腔体#3测试结果 1-OK  2-NG  3-腔体泄漏
LD TR0
ANDNOT W37.02  ; #3腔体抽真空异常结束
MOV(021) &2 D3156  ; 腔体#4测试结果 1-OK  2-NG  3-腔体泄漏
LD TR0
TIMX(550) 0456 &1  ; 检测异常传输

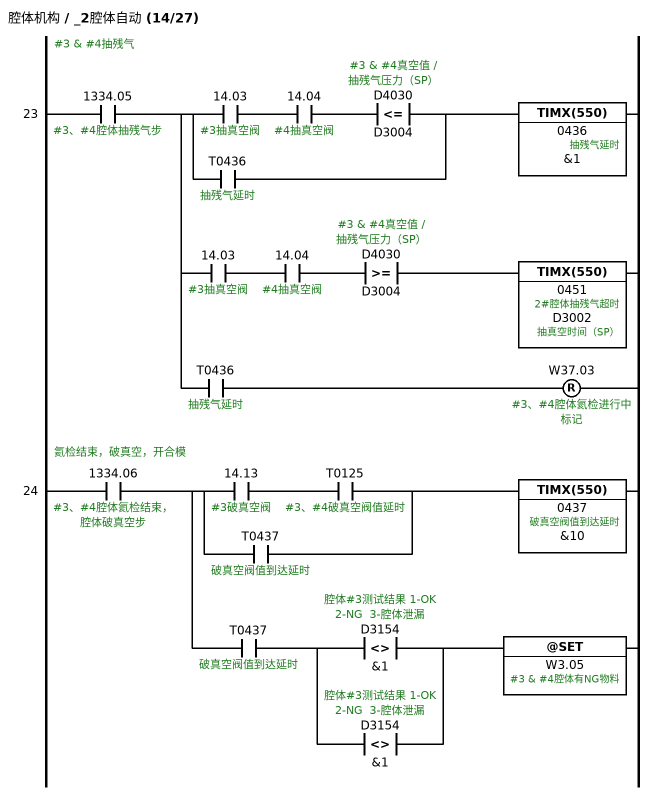
; rung 23: #3 & #4抽残气
LD 1334.05  ; #3、#4腔体抽残气步
OUT TR0
LD 14.03  ; #3抽真空阀
AND 14.04  ; #4抽真空阀
AND<=F(332) D4030 D3004  ; #3 & #4真空值, 抽残气压力（SP）
OR T0436  ; 抽残气延时
ANDLD
TIMX(550) 0436 &1  ; 抽残气延时
LD TR0
AND 14.03  ; #3抽真空阀
AND 14.04  ; #4抽真空阀
AND>=F(334) D4030 D3004  ; #3 & #4真空值, 抽残气压力（SP）
TIMX(550) 0451 D3002  ; 抽真空时间（SP）, 2#腔体抽残气超时
LD TR0
AND T0436  ; 抽残气延时
RSET W37.03  ; #3、#4腔体氦检进行中标记
; rung 24: 氦检结束，破真空，开合模
LD 1334.06  ; #3、#4腔体氦检结束，腔体破真空步
OUT TR0
LD 14.13  ; #3破真空阀
AND T0125  ; #3、#4破真空阀值延时
OR T0437  ; 破真空阀值到达延时
ANDLD
TIMX(550) 0437 &10  ; 破真空阀值到达延时
LD TR0
AND T0437  ; 破真空阀值到达延时
LD<>(305) D3154 &1  ; 腔体#3测试结果 1-OK  2-NG  3-腔体泄漏
OR<>(305) D3154 &1  ; 腔体#3测试结果 1-OK  2-NG  3-腔体泄漏
ANDLD
@SET W3.05  ; #3 & #4腔体有NG物料

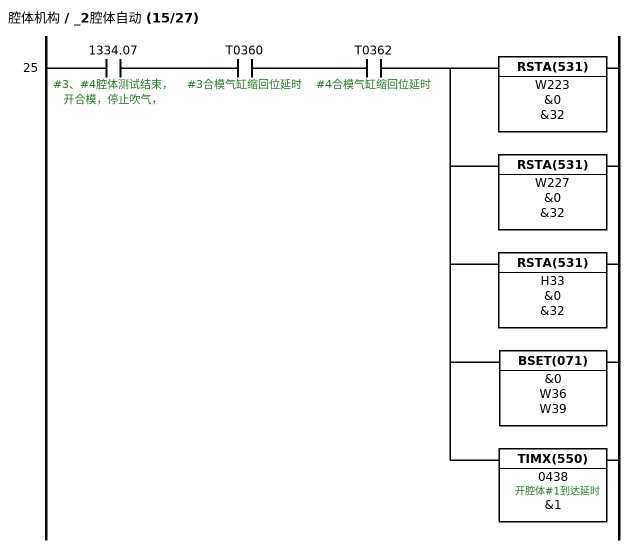
; rung 25
LD 1334.07  ; #3、#4腔体测试结束，开合模，停止吹气，
AND T0360  ; #3合模气缸缩回位延时
AND T0362  ; #4合模气缸缩回位延时
RSTA(531) W223 &0 &32
RSTA(531) W227 &0 &32
RSTA(531) H33 &0 &32
BSET(071) &0 W36 W39
TIMX(550) 0438 &1  ; 开腔体#1到达延时

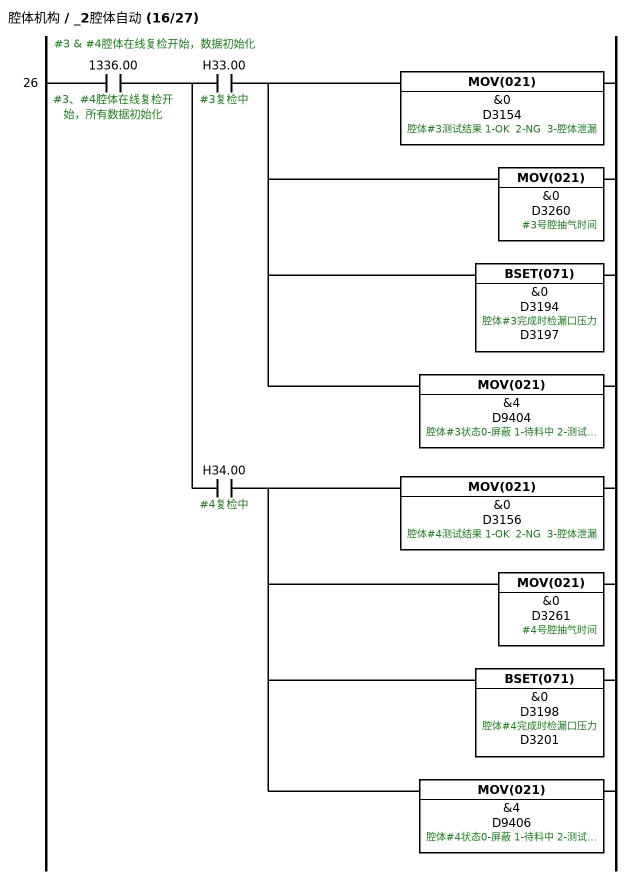
; rung 26: #3 & #4腔体在线复检开始，数据初始化
LD 1336.00  ; #3、#4腔体在线复检开始，所有数据初始化
OUT TR0
AND H33.00  ; #3复检中
MOV(021) &0 D3154  ; 腔体#3测试结果 1-OK  2-NG  3-腔体泄漏
MOV(021) &0 D3260  ; #3号腔抽气时间
BSET(071) &0 D3194 D3197  ; 腔体#3完成时检漏口压力
MOV(021) &4 D9404  ; 腔体#3状态0-屏蔽 1-待料中 2-测试中 3-测试完成 4-在线复检
LD TR0
AND H34.00  ; #4复检中
MOV(021) &0 D3156  ; 腔体#4测试结果 1-OK  2-NG  3-腔体泄漏
MOV(021) &0 D3261  ; #4号腔抽气时间
BSET(071) &0 D3198 D3201  ; 腔体#4完成时检漏口压力
MOV(021) &4 D9406  ; 腔体#4状态0-屏蔽 1-待料中 2-测试中 3-测试完成 4-在线复检

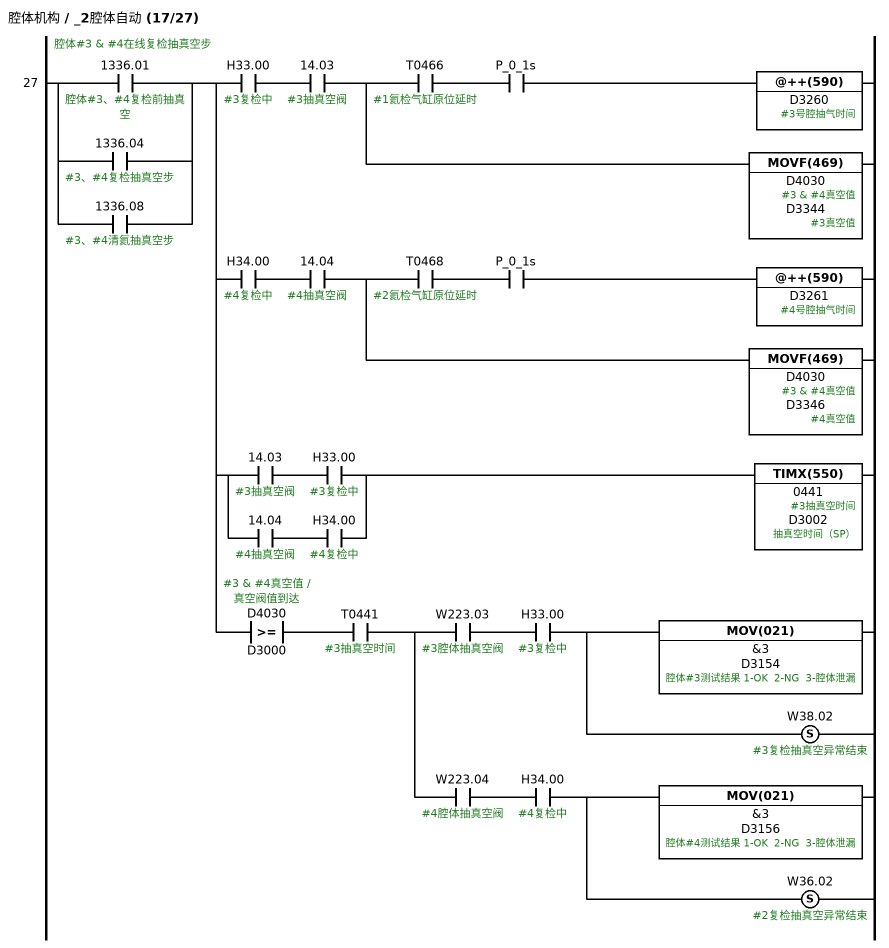
; rung 27: 腔体#3 & #4在线复检抽真空步
LD 1336.01  ; 腔体#3、#4复检前抽真空
OR 1336.04  ; #3、#4复检抽真空步
OR 1336.08  ; #3、#4清氦抽真空步
OUT TR0
AND H33.00  ; #3复检中
AND 14.03  ; #3抽真空阀
OUT TR1
AND T0466  ; #1氦检气缸原位延时
AND P_0_1s
@++(590) D3260  ; #3号腔抽气时间
LD TR1
MOVF(469) D4030 D3344  ; #3 & #4真空值, #3真空值
LD TR0
AND H34.00  ; #4复检中
AND 14.04  ; #4抽真空阀
OUT TR1
AND T0468  ; #2氦检气缸原位延时
AND P_0_1s
@++(590) D3261  ; #4号腔抽气时间
LD TR1
MOVF(469) D4030 D3346  ; #3 & #4真空值, #4真空值
LD TR0
LD 14.03  ; #3抽真空阀
AND H33.00  ; #3复检中
LD 14.04  ; #4抽真空阀
AND H34.00  ; #4复检中
ORLD
ANDLD
TIMX(550) 0441 D3002  ; 抽真空时间（SP）, #3抽真空时间
LD TR0
AND>=F(334) D4030 D3000  ; #3 & #4真空值, 真空阀值到达
AND T0441  ; #3抽真空时间
OUT TR0
AND W223.03  ; #3腔体抽真空阀
AND H33.00  ; #3复检中
MOV(021) &3 D3154  ; 腔体#3测试结果 1-OK  2-NG  3-腔体泄漏
SET W38.02  ; #3复检抽真空异常结束
LD TR0
AND W223.04  ; #4腔体抽真空阀
AND H34.00  ; #4复检中
MOV(021) &3 D3156  ; 腔体#4测试结果 1-OK  2-NG  3-腔体泄漏
SET W36.02  ; #2复检抽真空异常结束

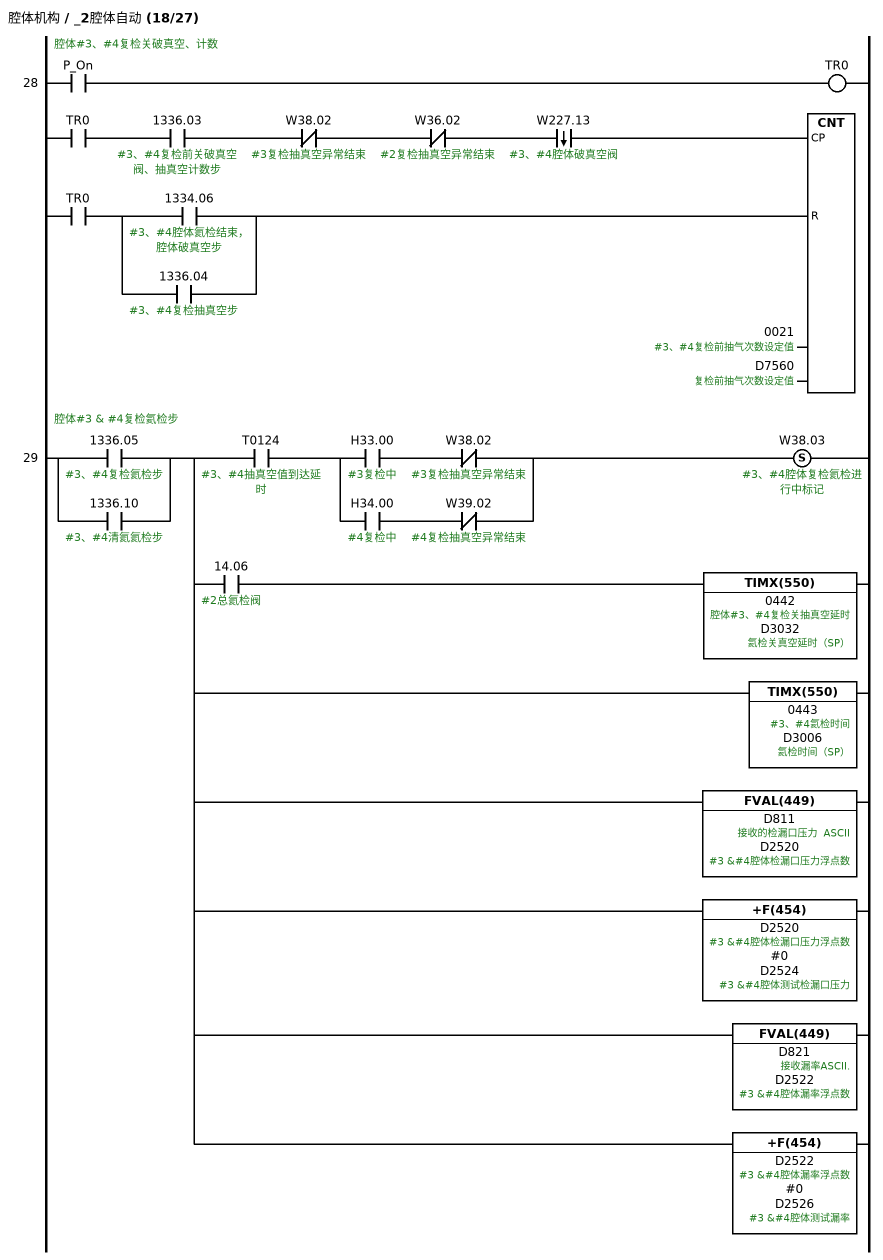
; rung 28: 腔体#3、#4复检关破真空、计数
LD P_On
OUT TR0
AND 1336.03  ; #3、#4复检前关破真空阀、抽真空计数步
ANDNOT W38.02  ; #3复检抽真空异常结束
ANDNOT W36.02  ; #2复检抽真空异常结束
%AND W227.13  ; #3、#4腔体破真空阀
LD TR0
LD 1334.06  ; #3、#4腔体氦检结束，腔体破真空步
OR 1336.04  ; #3、#4复检抽真空步
ANDLD
CNT 0021 D7560  ; 复检前抽气次数设定值, #3、#4复检前抽气次数设定值
; rung 29: 腔体#3 & #4复检氦检步
LD 1336.05  ; #3、#4复检氦检步
OR 1336.10  ; #3、#4清氦氦检步
OUT TR0
AND T0124  ; #3、#4抽真空值到达延时
LD H33.00  ; #3复检中
ANDNOT W38.02  ; #3复检抽真空异常结束
LD H34.00  ; #4复检中
ANDNOT W39.02  ; #4复检抽真空异常结束
ORLD
ANDLD
SET W38.03  ; #3、#4腔体复检氦检进行中标记
LD TR0
AND 14.06  ; #2总氦检阀
TIMX(550) 0442 D3032  ; 氦检关真空延时（SP）, 腔体#3、#4复检关抽真空延时
LD TR0
TIMX(550) 0443 D3006  ; 氦检时间（SP）, #3、#4氦检时间
FVAL(449) D811 D2520  ; 接收的检漏口压力  ASCII, #3 &#4腔体检漏口压力浮点数
+F(454) D2520 #0 D2524  ; #3 &#4腔体检漏口压力浮点数, #3 &#4腔体测试检漏口压力
FVAL(449) D821 D2522  ; 接收漏率ASCII., #3 &#4腔体漏率浮点数
+F(454) D2522 #0 D2526  ; #3 &#4腔体漏率浮点数, #3 &#4腔体测试漏率

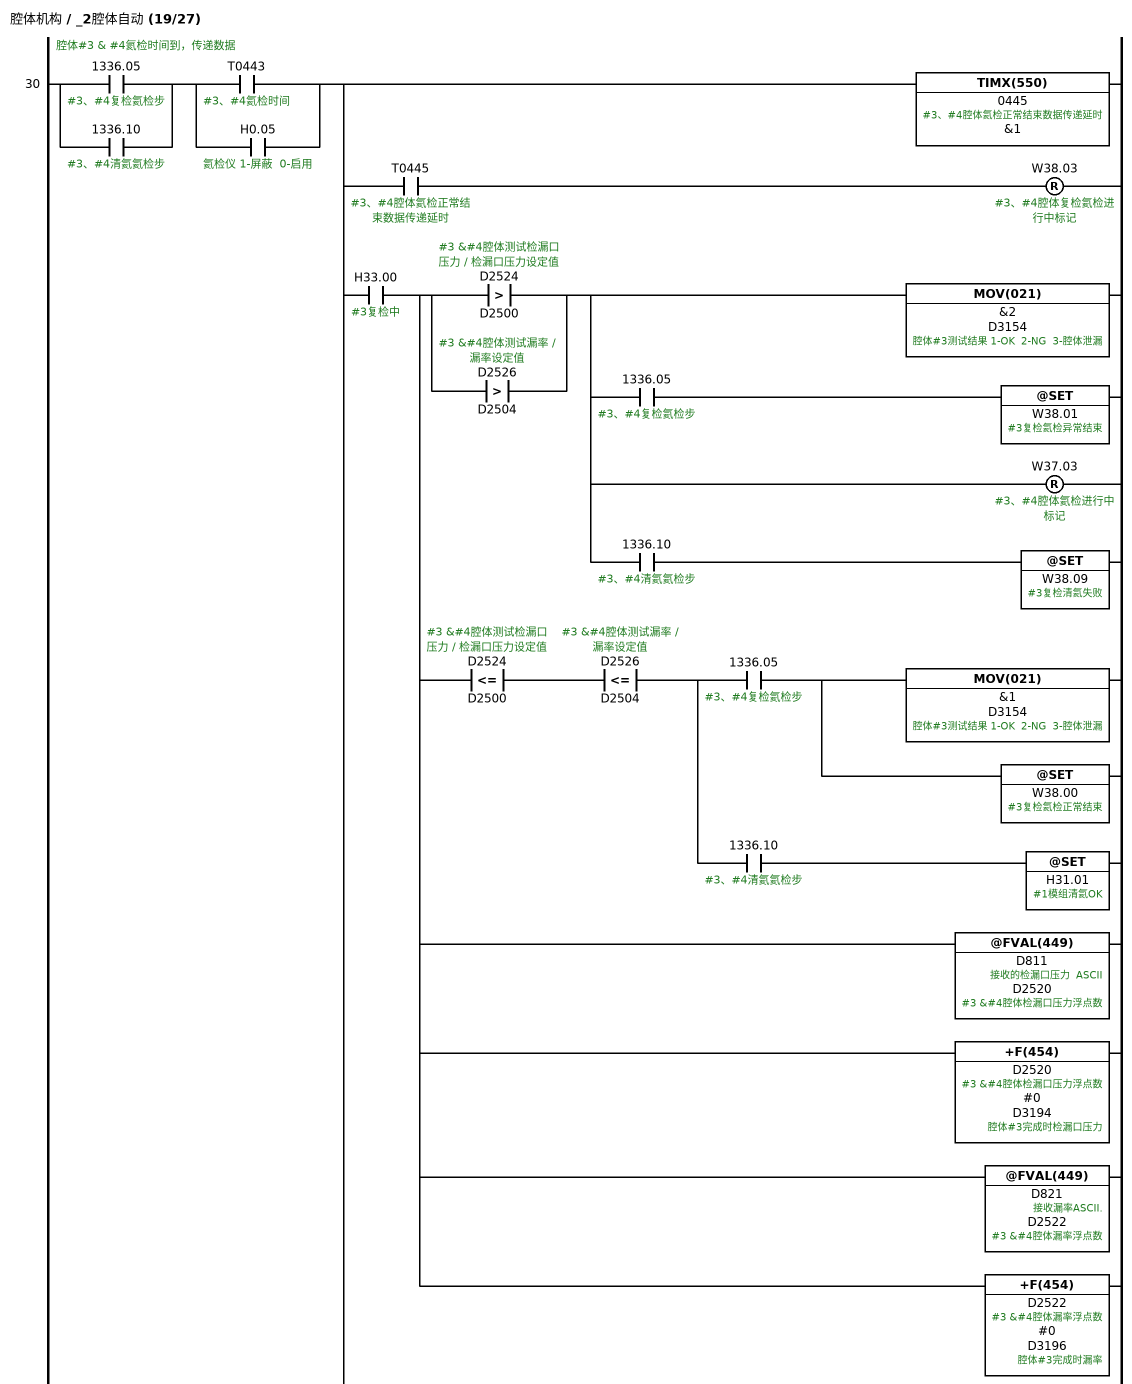

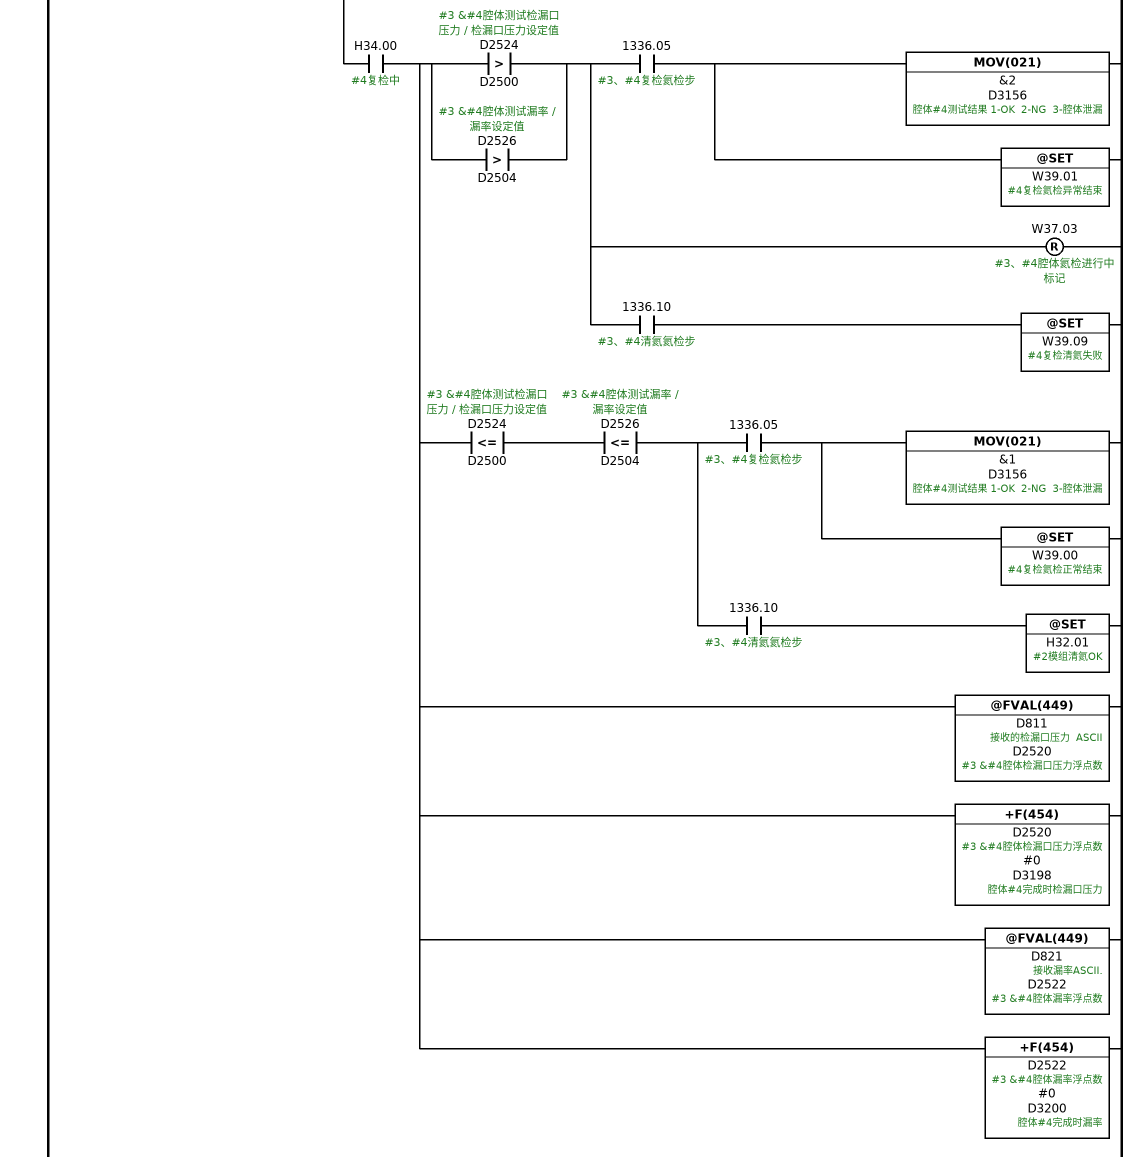
; rung 30: 腔体#3 & #4氦检时间到，传递数据
LD 1336.05  ; #3、#4复检氦检步
OR 1336.10  ; #3、#4清氦氦检步
LD T0443  ; #3、#4氦检时间
OR H0.05  ; 氦检仪 1-屏蔽  0-启用
ANDLD
OUT TR0
TIMX(550) 0445 &1  ; #3、#4腔体氦检正常结束数据传递延时
AND T0445  ; #3、#4腔体氦检正常结束数据传递延时
RSET W38.03  ; #3、#4腔体复检氦检进行中标记
LD TR0
AND H33.00  ; #3复检中
OUT TR1
LD>F(333) D2524 D2500  ; #3 &#4腔体测试检漏口压力, 检漏口压力设定值
OR>F(333) D2526 D2504  ; #3 &#4腔体测试漏率, 漏率设定值
ANDLD
OUT TR2
MOV(021) &2 D3154  ; 腔体#3测试结果 1-OK  2-NG  3-腔体泄漏
AND 1336.05  ; #3、#4复检氦检步
@SET W38.01  ; #3复检氦检异常结束
LD TR2
RSET W37.03  ; #3、#4腔体氦检进行中标记
AND 1336.10  ; #3、#4清氦氦检步
@SET W38.09  ; #3复检清氦失败
LD TR1
AND<=F(332) D2524 D2500  ; #3 &#4腔体测试检漏口压力, 检漏口压力设定值
AND<=F(332) D2526 D2504  ; #3 &#4腔体测试漏率, 漏率设定值
OUT TR2
AND 1336.05  ; #3、#4复检氦检步
MOV(021) &1 D3154  ; 腔体#3测试结果 1-OK  2-NG  3-腔体泄漏
@SET W38.00  ; #3复检氦检正常结束
LD TR2
AND 1336.10  ; #3、#4清氦氦检步
@SET H31.01  ; #1模组清氦OK
LD TR1
@FVAL(449) D811 D2520  ; 接收的检漏口压力  ASCII, #3 &#4腔体检漏口压力浮点数
+F(454) D2520 #0 D3194  ; #3 &#4腔体检漏口压力浮点数, 腔体#3完成时检漏口压力
@FVAL(449) D821 D2522  ; 接收漏率ASCII., #3 &#4腔体漏率浮点数
+F(454) D2522 #0 D3196  ; #3 &#4腔体漏率浮点数, 腔体#3完成时漏率
LD TR0
AND H34.00  ; #4复检中
OUT TR0
LD>F(333) D2524 D2500  ; #3 &#4腔体测试检漏口压力, 检漏口压力设定值
OR>F(333) D2526 D2504  ; #3 &#4腔体测试漏率, 漏率设定值
ANDLD
OUT TR1
AND 1336.05  ; #3、#4复检氦检步
MOV(021) &2 D3156  ; 腔体#4测试结果 1-OK  2-NG  3-腔体泄漏
@SET W39.01  ; #4复检氦检异常结束
LD TR1
RSET W37.03  ; #3、#4腔体氦检进行中标记
AND 1336.10  ; #3、#4清氦氦检步
@SET W39.09  ; #4复检清氦失败
LD TR0
AND<=F(332) D2524 D2500  ; #3 &#4腔体测试检漏口压力, 检漏口压力设定值
AND<=F(332) D2526 D2504  ; #3 &#4腔体测试漏率, 漏率设定值
OUT TR1
AND 1336.05  ; #3、#4复检氦检步
MOV(021) &1 D3156  ; 腔体#4测试结果 1-OK  2-NG  3-腔体泄漏
@SET W39.00  ; #4复检氦检正常结束
LD TR1
AND 1336.10  ; #3、#4清氦氦检步
@SET H32.01  ; #2模组清氦OK
LD TR0
@FVAL(449) D811 D2520  ; 接收的检漏口压力  ASCII, #3 &#4腔体检漏口压力浮点数
+F(454) D2520 #0 D3198  ; #3 &#4腔体检漏口压力浮点数, 腔体#4完成时检漏口压力
@FVAL(449) D821 D2522  ; 接收漏率ASCII., #3 &#4腔体漏率浮点数
+F(454) D2522 #0 D3200  ; #3 &#4腔体漏率浮点数, 腔体#4完成时漏率

